KUKA KRL program: MyProgram_309().src

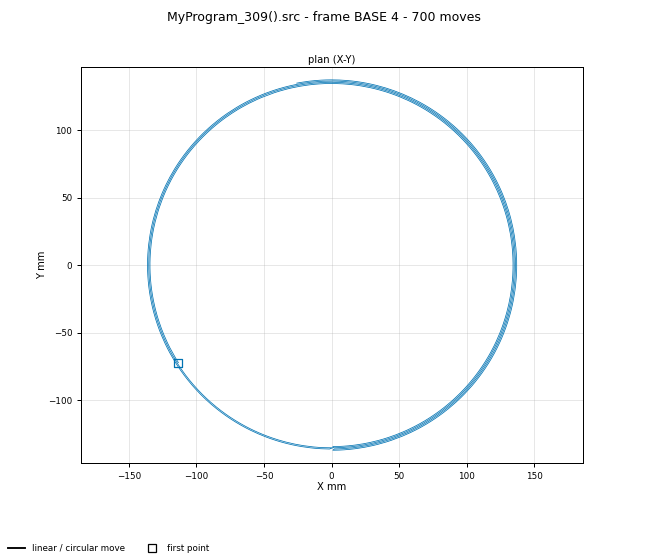
[picture p0: tool path of MyProgram_309().src in frame BASE 4, 700 of 700 moves have a stored position in this frame; points joined in program order, loops and branches not executed]
&ACCESS RVP
&REL 1
&PARAM TEMPLATE = C:\KRC\Roboter\Template\vorgabe
&PARAM EDITMASK = *
DEF MyProgram_309()
; ---- Setting reference (Base) ----
$BASE = BASE_DATA[4]

; --------------------------
; ---- Setting tool (TCP) ----
$TOOL = TOOL_DATA[3]
; --------------------------

$VEL.CP = VEL_APROX_PRINT
Startdeposition()
$VEL.CP = VEL_PRINT
LIN {X -113.3933,Y -72.2581,Z 182,A -144.0456,B 4.4589,C 0.2959,E1 4.3339,E2 236.7047} C_DIS
LIN {X -115.3766,Y -69.0471,Z 182,A -147.133,B 4.4585,C 0.3023,E1 4.3294,E2 239.9737} C_DIS
LIN {X -119.7006,Y -61.2412,Z 182,A -149.3934,B 4.4598,C 0.2824,E1 4.3266,E2 242.0427} C_DIS
LIN {X -121.551,Y -57.4829,Z 182,A -151.4804,B 4.46,C 0.28,E1 4.324,E2 244.1665} C_DIS
LIN {X -122.8459,Y -54.659,Z 182,A -152.8316,B 4.4602,C 0.2768,E1 4.3224,E2 245.5205} C_DIS
LIN {X -124.1948,Y -51.5211,Z 182,A -154.355,B 4.4604,C 0.2735,E1 4.3208,E2 247.0515} C_DIS
LIN {X -125.9546,Y -47.0544,Z 182,A -156.4644,B 4.4607,C 0.2686,E1 4.3186,E2 249.1678} C_DIS
LIN {X -127.2931,Y -43.3101,Z 182,A -158.1642,B 4.4609,C 0.2641,E1 4.3171,E2 250.8675} C_DIS
LIN {X -128.1422,Y -40.7223,Z 182,A -159.3873,B 4.4611,C 0.2614,E1 4.316,E2 252.0976} C_DIS
LIN {X -129.0534,Y -37.7348,Z 182,A -160.7492,B 4.4613,C 0.258,E1 4.3149,E2 253.4625} C_DIS
LIN {X -130.247,Y -33.3845,Z 182,A -162.5253,B 4.4616,C 0.2518,E1 4.3137,E2 255.2196} C_DIS
LIN {X -131.0025,Y -30.2853,Z 182,A -164.2358,B 4.4617,C 0.2504,E1 4.3125,E2 256.9725} C_DIS
LIN {X -131.9051,Y -26.083,Z 182,A -166.023,B 4.462,C 0.2451,E1 4.3115,E2 258.7533} C_DIS
LIN {X -132.6145,Y -22.1846,Z 182,A -167.7411,B 4.4623,C 0.2406,E1 4.3107,E2 260.4739} C_DIS
LIN {X -133.1933,Y -18.4034,Z 182,A -169.5897,B 4.4624,C 0.2374,E1 4.3099,E2 262.3483} C_DIS
LIN {X -133.6998,Y -14.2533,Z 182,A -171.2997,B 4.4627,C 0.2319,E1 4.3094,E2 264.0484} C_DIS
LIN {X -134.0654,Y -10.2705,Z 182,A -173.1645,B 4.4629,C 0.2282,E1 4.3089,E2 265.9317} C_DIS
LIN {X -134.3281,Y -5.9384,Z 182,A -174.9356,B 4.4632,C 0.2224,E1 4.3087,E2 267.6919} C_DIS
LIN {X -134.4379,Y -2.2975,Z 182,A -176.6146,B 4.4634,C 0.2188,E1 4.3085,E2 269.3853} C_DIS
LIN {X -134.4464,Y 1.7844,Z 182,A -178.4359,B 4.4636,C 0.2144,E1 4.3085,E2 271.2154} C_DIS
LIN {X -134.354,Y 5.2733,Z 182,A -179.936,B 4.4638,C 0.2103,E1 4.3087,E2 272.716} C_DIS
LIN {X -134.1215,Y 9.5026,Z 182,A 178.1862,B 4.464,C 0.2057,E1 4.309,E2 274.6013} C_DIS
LIN {X -133.8199,Y 13.0792,Z 182,A 176.6504,B 4.4642,C 0.2014,E1 4.3094,E2 276.1368} C_DIS
LIN {X -133.502,Y 15.9997,Z 182,A 175.3587,B 4.4643,C 0.1981,E1 4.3098,E2 277.4323} C_DIS
LIN {X -133.023,Y 19.5953,Z 182,A 173.6191,B 4.4645,C 0.195,E1 4.3105,E2 279.1944} C_DIS
LIN {X -132.3689,Y 23.6053,Z 182,A 171.9298,B 4.4647,C 0.1899,E1 4.3113,E2 280.8772} C_DIS
LIN {X -131.671,Y 27.2336,Z 182,A 170.256,B 4.4649,C 0.1861,E1 4.3122,E2 282.5618} C_DIS
LIN {X -130.5324,Y 32.2586,Z 182,A 168.0955,B 4.4651,C 0.1799,E1 4.3136,E2 284.7163} C_DIS
LIN {X -129.2234,Y 37.1542,Z 182,A 165.915,B 4.4653,C 0.1741,E1 4.3152,E2 286.8977} C_DIS
LIN {X -128.5071,Y 39.5558,Z 182,A 164.7164,B 4.4654,C 0.172,E1 4.3162,E2 288.1112} C_DIS
LIN {X -127.5833,Y 42.4406,Z 182,A 163.3928,B 4.4655,C 0.1687,E1 4.3173,E2 289.4377} C_DIS
LIN {X -126.1534,Y 46.5237,Z 182,A 161.5675,B 4.4657,C 0.1637,E1 4.319,E2 291.2594} C_DIS
LIN {X -125.1691,Y 49.1075,Z 182,A 160.3104,B 4.4658,C 0.1611,E1 4.3203,E2 292.525} C_DIS
LIN {X -123.9551,Y 52.095,Z 182,A 158.8275,B 4.4659,C 0.1582,E1 4.3219,E2 294.0197} C_DIS
LIN {X -122.5618,Y 55.2941,Z 182,A 157.3536,B 4.4661,C 0.1543,E1 4.3236,E2 295.4909} C_DIS
LIN {X -121.0569,Y 58.5172,Z 182,A 155.4896,B 4.4661,C 0.1527,E1 4.3259,E2 297.3955} C_DIS
LIN {X -118.7591,Y 63.0499,Z 182,A 153.5389,B 4.4664,C 0.1458,E1 4.3283,E2 299.3186} C_DIS
LIN {X -116.7267,Y 66.7391,Z 182,A 151.5986,B 4.4664,C 0.1424,E1 4.331,E2 301.275} C_DIS
LIN {X -114.4006,Y 70.6531,Z 182,A 149.1045,B 4.4664,C 0.1414,E1 4.3347,E2 303.8333} C_DIS
LIN {X -111.8542,Y 74.6179,Z 182,A 147.5238,B 4.4667,C 0.1338,E1 4.3371,E2 305.3616} C_DIS
LIN {X -109.1703,Y 78.493,Z 182,A 145.5025,B 4.4669,C 0.1293,E1 4.3403,E2 307.3828} C_DIS
LIN {X -106.7613,Y 81.7387,Z 182,A 143.725,B 4.4669,C 0.1258,E1 4.3433,E2 309.1654} C_DIS
LIN {X -104.0626,Y 85.1479,Z 182,A 141.8241,B 4.4671,C 0.122,E1 4.3467,E2 311.0705} C_DIS
LIN {X -101.1349,Y 88.6059,Z 182,A 139.8527,B 4.4671,C 0.1182,E1 4.3503,E2 313.0452} C_DIS
LIN {X -98.1961,Y 91.8521,Z 182,A 137.9249,B 4.4673,C 0.1148,E1 4.3539,E2 314.9788} C_DIS
LIN {X -95.323,Y 94.83,Z 182,A 136.1391,B 4.4673,C 0.1114,E1 4.3574,E2 316.7659} C_DIS
LIN {X -92.1703,Y 97.8971,Z 182,A 134.199,B 4.4674,C 0.1083,E1 4.3613,E2 318.7124} C_DIS
LIN {X -88.8308,Y 100.9375,Z 182,A 132.2757,B 4.4675,C 0.1047,E1 4.3653,E2 320.634} C_DIS
LIN {X -85.661,Y 103.6407,Z 182,A 130.4375,B 4.4675,C 0.102,E1 4.3693,E2 322.4783} C_DIS
LIN {X -82.322,Y 106.3122,Z 182,A 128.5912,B 4.4676,C 0.099,E1 4.3733,E2 324.3259} C_DIS
LIN {X -78.8871,Y 108.8854,Z 182,A 126.7591,B 4.4676,C 0.096,E1 4.3775,E2 326.1571} C_DIS
LIN {X -73.7106,Y 112.4545,Z 182,A 123.4758,B 4.4676,C 0.0965,E1 4.3852,E2 329.5096} C_DIS
LIN {X -69.7248,Y 114.9682,Z 182,A 122.124,B 4.4679,C 0.0886,E1 4.3883,E2 330.7825} C_DIS
LIN {X -66.9003,Y 116.6347,Z 182,A 120.1078,B 4.4678,C 0.0914,E1 4.3933,E2 332.8708} C_DIS
LIN {X -63.1989,Y 118.6809,Z 182,A 118.798,B 4.4679,C 0.0852,E1 4.3964,E2 334.1213} C_DIS
LIN {X -61.0835,Y 119.7809,Z 182,A 117.6379,B 4.4679,C 0.0852,E1 4.3993,E2 335.2977} C_DIS
LIN {X -57.3839,Y 121.5983,Z 182,A 115.9821,B 4.4679,C 0.0822,E1 4.4034,E2 336.9403} C_DIS
LIN {X -54.881,Y 122.7466,Z 182,A 114.6943,B 4.4679,C 0.0818,E1 4.4068,E2 338.2408} C_DIS
LIN {X -51.5957,Y 124.1636,Z 182,A 113.1875,B 4.468,C 0.0801,E1 4.4106,E2 339.7446} C_DIS
LIN {X -42.4267,Y 127.5879,Z 182,A 108.5492,B 4.468,C 0.0801,E1 4.423,E2 344.4352} C_DIS
LIN {X -38.4167,Y 128.8538,Z 182,A 107.2755,B 4.4681,C 0.0745,E1 4.4262,E2 345.6469} C_DIS
LIN {X -35.4991,Y 129.6884,Z 182,A 105.9279,B 4.4681,C 0.074,E1 4.4298,E2 347.0002} C_DIS
LIN {X -32.7166,Y 130.4165,Z 182,A 104.7062,B 4.4681,C 0.0732,E1 4.4331,E2 348.2206} C_DIS
LIN {X -29.8649,Y 131.0985,Z 182,A 103.3874,B 4.4681,C 0.0731,E1 4.4367,E2 349.5468} C_DIS
LIN {X -26.0554,Y 131.9107,Z 182,A 101.7586,B 4.4681,C 0.0719,E1 4.4412,E2 351.1712} C_DIS
LIN {X -23.3572,Y 132.4133,Z 182,A 100.6147,B 4.4681,C 0.0712,E1 4.4443,E2 352.3113} C_DIS
LIN {X -19.9287,Y 132.9738,Z 182,A 99.0996,B 4.4681,C 0.071,E1 4.4485,E2 353.8298} C_DIS
LIN {X -16.7934,Y 133.4062,Z 182,A 97.2359,B 4.4681,C 0.0751,E1 4.4538,E2 355.7534} C_DIS
LIN {X -12.6819,Y 133.858,Z 182,A 95.9309,B 4.4681,C 0.0707,E1 4.4573,E2 357.0037} C_DIS
LIN {X -9.5581,Y 134.1174,Z 182,A 94.5437,B 4.4681,C 0.0709,E1 4.4612,E2 358.3963} C_DIS
LIN {X -5.5166,Y 134.3445,Z 182,A 92.8589,B 4.4681,C 0.0704,E1 4.4659,E2 360.0755} C_DIS
LIN {X -1.4978,Y 134.4505,Z 182,A 91.015,B 4.4681,C 0.0717,E1 4.4711,E2 361.9342} C_DIS
LIN {X 2.3924,Y 134.4363,Z 182,A 89.4627,B 4.4681,C 0.0708,E1 4.4754,E2 363.4733} C_DIS
LIN {X 5.8114,Y 134.333,Z 182,A 88.1347,B 4.4681,C 0.0699,E1 4.479,E2 364.7854} C_DIS
LIN {X 8.5441,Y 134.1859,Z 182,A 86.7961,B 4.4681,C 0.0718,E1 4.4828,E2 366.1439} C_DIS
LIN {X 13.4353,Y 133.7857,Z 182,A 84.7941,B 4.4681,C 0.0716,E1 4.4884,E2 368.1346} C_DIS
LIN {X 17.4287,Y 133.3229,Z 182,A 83.0133,B 4.4681,C 0.0729,E1 4.4933,E2 369.9227} C_DIS
LIN {X 22.1823,Y 132.6148,Z 182,A 81.0965,B 4.4681,C 0.0727,E1 4.4986,E2 371.8234} C_DIS
LIN {X 25.2731,Y 132.0606,Z 182,A 79.7667,B 4.4681,C 0.0734,E1 4.5022,E2 373.1518} C_DIS
LIN {X 28.5205,Y 131.3976,Z 182,A 78.3441,B 4.4681,C 0.0744,E1 4.5061,E2 374.5753} C_DIS
LIN {X 32.4205,Y 130.4917,Z 182,A 76.5461,B 4.4681,C 0.0765,E1 4.511,E2 376.3837} C_DIS
LIN {X 36.0959,Y 129.5215,Z 182,A 74.531,B 4.468,C 0.0819,E1 4.5166,E2 378.445} C_DIS
LIN {X 40.4003,Y 128.2448,Z 182,A 73.2819,B 4.468,C 0.0768,E1 4.5197,E2 379.6153} C_DIS
LIN {X 43.736,Y 127.1454,Z 182,A 71.5814,B 4.468,C 0.0803,E1 4.5243,E2 381.3396} C_DIS
LIN {X 47.3865,Y 125.8303,Z 182,A 70.0326,B 4.468,C 0.0809,E1 4.5283,E2 382.8757} C_DIS
LIN {X 50.52,Y 124.6053,Z 182,A 68.6167,B 4.468,C 0.0823,E1 4.532,E2 384.2893} C_DIS
LIN {X 54.1914,Y 123.0551,Z 182,A 66.9764,B 4.468,C 0.0837,E1 4.5362,E2 385.9226} C_DIS
LIN {X 56.6157,Y 121.9564,Z 182,A 65.8155,B 4.468,C 0.0854,E1 4.5391,E2 387.0865} C_DIS
LIN {X 59.7801,Y 120.4371,Z 182,A 64.3292,B 4.4679,C 0.0872,E1 4.5428,E2 388.5715} C_DIS
LIN {X 63.1887,Y 118.6862,Z 182,A 62.8242,B 4.4679,C 0.0881,E1 4.5465,E2 390.0613} C_DIS
LIN {X 66.3073,Y 116.9729,Z 182,A 61.1293,B 4.4678,C 0.0922,E1 4.5507,E2 391.7774} C_DIS
LIN {X 69.8955,Y 114.8649,Z 182,A 59.4108,B 4.4678,C 0.0943,E1 4.5548,E2 393.4893} C_DIS
LIN {X 73.1101,Y 112.8456,Z 182,A 57.8239,B 4.4677,C 0.0964,E1 4.5586,E2 395.0726} C_DIS
LIN {X 76.8735,Y 110.3162,Z 182,A 55.9392,B 4.4677,C 0.0991,E1 4.5629,E2 396.9517} C_DIS
LIN {X 80.1605,Y 107.9515,Z 182,A 54.2252,B 4.4676,C 0.1019,E1 4.5667,E2 398.6644} C_DIS
LIN {X 83.4929,Y 105.3956,Z 182,A 52.5057,B 4.4676,C 0.1043,E1 4.5705,E2 400.3757} C_DIS
LIN {X 86.7231,Y 102.7543,Z 182,A 50.7346,B 4.4674,C 0.1075,E1 4.5743,E2 402.1461} C_DIS
LIN {X 90.7436,Y 99.2215,Z 182,A 48.5047,B 4.4674,C 0.1113,E1 4.579,E2 404.3703} C_DIS
LIN {X 93.9259,Y 96.2144,Z 182,A 46.66,B 4.4673,C 0.1148,E1 4.5827,E2 406.2127} C_DIS
LIN {X 97.2485,Y 92.8543,Z 182,A 44.8621,B 4.4673,C 0.1164,E1 4.5861,E2 407.9851} C_DIS
LIN {X 99.7983,Y 90.1088,Z 182,A 43.1522,B 4.4671,C 0.1211,E1 4.5894,E2 409.709} C_DIS
LIN {X 102.7253,Y 86.7572,Z 182,A 41.3372,B 4.4671,C 0.1243,E1 4.5927,E2 411.5147} C_DIS
LIN {X 105.486,Y 83.379,Z 182,A 39.4855,B 4.4669,C 0.1283,E1 4.5959,E2 413.366} C_DIS
LIN {X 107.6526,Y 80.5619,Z 182,A 38.1164,B 4.4669,C 0.13,E1 4.5982,E2 414.718} C_DIS
LIN {X 110.0357,Y 77.2749,Z 182,A 36.3306,B 4.4667,C 0.1347,E1 4.6011,E2 416.5112} C_DIS
LIN {X 112.198,Y 74.1002,Z 182,A 34.758,B 4.4667,C 0.1378,E1 4.6035,E2 418.0765} C_DIS
LIN {X 114.3595,Y 70.7194,Z 182,A 33.0845,B 4.4665,C 0.1415,E1 4.606,E2 419.7462} C_DIS
LIN {X 116.2486,Y 67.5685,Z 182,A 31.557,B 4.4664,C 0.1449,E1 4.6082,E2 421.2697} C_DIS
LIN {X 118.4291,Y 63.6691,Z 182,A 29.7729,B 4.4663,C 0.1482,E1 4.6106,E2 423.0401} C_DIS
LIN {X 119.8546,Y 60.9386,Z 182,A 28.4894,B 4.4662,C 0.1511,E1 4.6122,E2 424.3205} C_DIS
LIN {X 121.6394,Y 57.298,Z 182,A 26.8491,B 4.4661,C 0.1545,E1 4.6142,E2 425.951} C_DIS
LIN {X 122.7451,Y 54.8845,Z 182,A 25.7578,B 4.466,C 0.1569,E1 4.6154,E2 427.0379} C_DIS
LIN {X 124.9219,Y 49.7342,Z 182,A 23.1326,B 4.4656,C 0.1662,E1 4.6182,E2 429.6938} C_DIS
LIN {X 126.1191,Y 46.6154,Z 182,A 22.0493,B 4.4656,C 0.1657,E1 4.6193,E2 430.7365} C_DIS
LIN {X 127.1406,Y 43.7499,Z 182,A 20.7434,B 4.4656,C 0.1693,E1 4.6205,E2 432.0441} C_DIS
LIN {X 128.3104,Y 40.1957,Z 182,A 19.2597,B 4.4654,C 0.1722,E1 4.6217,E2 433.5152} C_DIS
LIN {X 129.3835,Y 36.5893,Z 182,A 17.6578,B 4.4652,C 0.1766,E1 4.623,E2 435.1177} C_DIS
LIN {X 130.3423,Y 33.0092,Z 182,A 16.1637,B 4.4652,C 0.1798,E1 4.624,E2 436.6024} C_DIS
LIN {X 131.1561,Y 29.6128,Z 182,A 14.671,B 4.4649,C 0.184,E1 4.625,E2 438.0965} C_DIS
LIN {X 131.8816,Y 26.1986,Z 182,A 13.2924,B 4.4649,C 0.1868,E1 4.6257,E2 439.4627} C_DIS
LIN {X 132.435,Y 23.2362,Z 182,A 12.0709,B 4.4647,C 0.1896,E1 4.6263,E2 440.6772} C_DIS
LIN {X 132.9509,Y 20.0765,Z 182,A 10.6053,B 4.4645,C 0.1947,E1 4.627,E2 442.1561} C_DIS
LIN {X 133.4213,Y 16.6763,Z 182,A 9.3253,B 4.4645,C 0.1965,E1 4.6274,E2 443.4147} C_DIS
LIN {X 133.7277,Y 13.9936,Z 182,A 8.2364,B 4.4643,C 0.1989,E1 4.6278,E2 444.4967} C_DIS
LIN {X 134.0514,Y 10.4624,Z 182,A 6.6919,B 4.4641,C 0.2036,E1 4.6281,E2 446.0464} C_DIS
LIN {X 134.3161,Y 6.1891,Z 182,A 4.7647,B 4.4638,C 0.2101,E1 4.6284,E2 447.9875} C_DIS
LIN {X 134.4515,Y 1.4573,Z 182,A 2.9283,B 4.4636,C 0.2135,E1 4.6285,E2 449.8031} C_DIS
LIN {X 134.4277,Y -2.9093,Z 182,A 1.2197,B 4.4635,C 0.2169,E1 4.6285,E2 451.4941} C_DIS
LIN {X 134.2584,Y -7.3369,Z 182,A -0.614,B 4.4632,C 0.2215,E1 4.6283,E2 453.3225} C_DIS
LIN {X 133.9862,Y -11.2465,Z 182,A -2.334,B 4.463,C 0.2269,E1 4.6279,E2 455.0498} C_DIS
LIN {X 133.6364,Y -14.8426,Z 182,A -3.7012,B 4.4629,C 0.229,E1 4.6275,E2 456.3969} C_DIS
LIN {X 133.2626,Y -17.8893,Z 182,A -5.1369,B 4.4626,C 0.2344,E1 4.627,E2 457.8494} C_DIS
LIN {X 132.5488,Y -22.5782,Z 182,A -6.9217,B 4.4624,C 0.237,E1 4.6262,E2 459.6064} C_DIS
LIN {X 131.9195,Y -26.0115,Z 182,A -8.3947,B 4.4622,C 0.241,E1 4.6254,E2 461.0789} C_DIS
LIN {X 131.2851,Y -29.0417,Z 182,A -9.6737,B 4.4621,C 0.2442,E1 4.6247,E2 462.3539} C_DIS
LIN {X 130.6233,Y -31.8813,Z 182,A -10.8534,B 4.4619,C 0.2468,E1 4.6239,E2 463.5267} C_DIS
LIN {X 129.8554,Y -34.8762,Z 182,A -12.2063,B 4.4617,C 0.2509,E1 4.623,E2 464.8851} C_DIS
LIN {X 128.6748,Y -39.008,Z 182,A -13.9853,B 4.4614,C 0.2553,E1 4.6216,E2 466.6591} C_DIS
LIN {X 127.1875,Y -43.6146,Z 182,A -15.9399,B 4.4612,C 0.2595,E1 4.6199,E2 468.6019} C_DIS
LIN {X 126.027,Y -46.8614,Z 182,A -17.5288,B 4.4609,C 0.2649,E1 4.6183,E2 470.2069} C_DIS
LIN {X 124.5326,Y -50.7002,Z 182,A -19.1914,B 4.4607,C 0.2684,E1 4.6166,E2 471.8594} C_DIS
LIN {X 123.1292,Y -54.0221,Z 182,A -20.5599,B 4.4606,C 0.2704,E1 4.6151,E2 473.2082} C_DIS
LIN {X 121.8799,Y -56.7812,Z 182,A -21.9042,B 4.4603,C 0.2744,E1 4.6136,E2 474.5602} C_DIS
LIN {X 120.3627,Y -59.9308,Z 182,A -23.2834,B 4.4602,C 0.2769,E1 4.6119,E2 475.9268} C_DIS
LIN {X 118.0655,Y -64.3408,Z 182,A -25.3175,B 4.4599,C 0.2812,E1 4.6092,E2 477.9522} C_DIS
LIN {X 116.1605,Y -67.7206,Z 182,A -27.0291,B 4.4596,C 0.2861,E1 4.6069,E2 479.6725} C_DIS
LIN {X 114.0228,Y -71.2606,Z 182,A -28.7623,B 4.4593,C 0.29,E1 4.6043,E2 481.4035} C_DIS
LIN {X 111.6949,Y -74.8566,Z 182,A -30.5206,B 4.4591,C 0.2936,E1 4.6016,E2 483.155} C_DIS
LIN {X 109.3703,Y -78.2134,Z 182,A -32.2078,B 4.4589,C 0.2971,E1 4.5989,E2 484.837} C_DIS
LIN {X 106.689,Y -81.8333,Z 182,A -34.0857,B 4.4586,C 0.301,E1 4.5958,E2 486.7113} C_DIS
LIN {X 104.0053,Y -85.2181,Z 182,A -35.8735,B 4.4584,C 0.3046,E1 4.5927,E2 488.494} C_DIS
LIN {X 100.7335,Y -89.0616,Z 182,A -37.7925,B 4.4582,C 0.3065,E1 4.5892,E2 490.3856} C_DIS
LIN {X 98.2774,Y -91.7648,Z 182,A -39.4623,B 4.4579,C 0.3112,E1 4.586,E2 492.071} C_DIS
LIN {X 95.1977,Y -94.9561,Z 182,A -41.3675,B 4.4576,C 0.3154,E1 4.5823,E2 493.9798} C_DIS
LIN {X 91.2794,Y -98.729,Z 182,A -43.4698,B 4.4575,C 0.3175,E1 4.5781,E2 496.0567} C_DIS
LIN {X 88.6795,Y -101.0706,Z 182,A -45.1059,B 4.4571,C 0.3222,E1 4.5746,E2 497.7125} C_DIS
LIN {X 85.3767,Y -103.8756,Z 182,A -46.8502,B 4.457,C 0.3245,E1 4.5709,E2 499.4453} C_DIS
LIN {X 82.3404,Y -106.298,Z 182,A -48.4788,B 4.4568,C 0.3272,E1 4.5673,E2 501.0719} C_DIS
LIN {X 79.5563,Y -108.3974,Z 182,A -49.8643,B 4.4566,C 0.3287,E1 4.5643,E2 502.4459} C_DIS
LIN {X 76.4279,Y -110.6261,Z 182,A -51.562,B 4.4564,C 0.3322,E1 4.5604,E2 504.1526} C_DIS
LIN {X 72.8163,Y -113.0359,Z 182,A -53.3398,B 4.4562,C 0.3344,E1 4.5562,E2 505.9227} C_DIS
LIN {X 69.2003,Y -115.2851,Z 182,A -55.1591,B 4.456,C 0.3373,E1 4.5519,E2 507.744} C_DIS
LIN {X 65.4541,Y -117.4525,Z 182,A -56.9794,B 4.4558,C 0.3398,E1 4.5475,E2 509.5626} C_DIS
LIN {X 61.3924,Y -119.6236,Z 182,A -58.6597,B 4.4558,C 0.3394,E1 4.5434,E2 511.2085} C_DIS
LIN {X 58.673,Y -120.9825,Z 182,A -60.0649,B 4.4556,C 0.3424,E1 4.5398,E2 512.6287} C_DIS
LIN {X 56.3839,Y -122.0636,Z 182,A -61.2344,B 4.4554,C 0.3449,E1 4.5369,E2 513.8104} C_DIS
LIN {X 52.8908,Y -123.6183,Z 182,A -63.5089,B 4.4547,C 0.3541,E1 4.5308,E2 516.1677} C_DIS
LIN {X 47.5793,Y -125.7581,Z 182,A -65.014,B 4.4553,C 0.3465,E1 4.5272,E2 517.5561} C_DIS
LIN {X 42.1713,Y -127.6729,Z 182,A -67.5798,B 4.455,C 0.3505,E1 4.5204,E2 520.1391} C_DIS
LIN {X 38.1773,Y -128.9239,Z 182,A -69.4257,B 4.4548,C 0.3528,E1 4.5154,E2 521.9942} C_DIS
LIN {X 34.3309,Y -130.0008,Z 182,A -71.0744,B 4.4548,C 0.3537,E1 4.511,E2 523.6372} C_DIS
LIN {X 30.9344,Y -130.8515,Z 182,A -72.4808,B 4.4548,C 0.354,E1 4.5072,E2 525.0336} C_DIS
LIN {X 28.1939,Y -131.4681,Z 182,A -73.6699,B 4.4546,C 0.3548,E1 4.5039,E2 526.2224} C_DIS
LIN {X 23.3364,Y -132.4171,Z 182,A -75.7501,B 4.4546,C 0.3559,E1 4.4983,E2 528.3002} C_DIS
LIN {X 19.8941,Y -132.9791,Z 182,A -77.228,B 4.4546,C 0.3567,E1 4.4942,E2 529.778} C_DIS
LIN {X 17.3536,Y -133.3328,Z 182,A -78.4563,B 4.4543,C 0.3586,E1 4.4907,E2 531.024} C_DIS
LIN {X 12.3919,Y -133.8859,Z 182,A -80.9068,B 4.454,C 0.3628,E1 4.4838,E2 533.5168} C_DIS
LIN {X 8.4264,Y -134.1932,Z 182,A -82.1981,B 4.4543,C 0.3593,E1 4.4803,E2 534.7576} C_DIS
LIN {X 4.743,Y -134.3747,Z 182,A -83.6718,B 4.4543,C 0.3587,E1 4.4762,E2 536.2197} C_DIS
LIN {X 0.9641,Y -134.4524,Z 182,A -85.5454,B 4.4541,C 0.3616,E1 4.4709,E2 538.1275} C_DIS
Enddeposition()
LIN {X 0.9641,Y -134.4524,Z 182,A -85.5454,B 4.4541,C 0.3616,E1 4.4709,E2 538.1275} C_DIS
Startdeposition()
$VEL.CP = VEL_PRINT
LIN {X 1.5996,Y -135.3511,Z 182,A -84.3043,B 4.4548,C 0.3542,E1 4.4748,E2 536.7934} C_DIS
LIN {X 8.4271,Y -135.0963,Z 182,A -81.4838,B 4.4548,C 0.3542,E1 4.4826,E2 533.9808} C_DIS
LIN {X 15.2303,Y -134.5013,Z 182,A -78.6391,B 4.4548,C 0.3535,E1 4.4905,E2 531.1406} C_DIS
LIN {X 18.8912,Y -134.0342,Z 182,A -77.0659,B 4.4548,C 0.3526,E1 4.4948,E2 529.5651} C_DIS
LIN {X 23.0843,Y -133.378,Z 182,A -75.0501,B 4.4552,C 0.3492,E1 4.5005,E2 527.5198} C_DIS
LIN {X 28.2212,Y -132.3845,Z 182,A -73.118,B 4.455,C 0.3507,E1 4.5057,E2 525.623} C_DIS
LIN {X 31.6043,Y -131.6174,Z 182,A -71.686,B 4.455,C 0.35,E1 4.5095,E2 524.1948} C_DIS
LIN {X 34.9586,Y -130.7664,Z 182,A -70.192,B 4.4552,C 0.3484,E1 4.5136,E2 522.6961} C_DIS
LIN {X 38.6291,Y -129.7309,Z 182,A -68.4986,B 4.4554,C 0.3461,E1 4.5182,E2 520.9914} C_DIS
LIN {X 42.4486,Y -128.5307,Z 182,A -66.9042,B 4.4554,C 0.3455,E1 4.5224,E2 519.4089} C_DIS
LIN {X 46.6809,Y -127.057,Z 182,A -64.7935,B 4.4558,C 0.341,E1 4.528,E2 517.2691} C_DIS
LIN {X 53.5716,Y -124.3061,Z 182,A -61.9854,B 4.4558,C 0.341,E1 4.5352,E2 514.5021} C_DIS
LIN {X 56.4713,Y -123.0164,Z 182,A -60.6059,B 4.4559,C 0.339,E1 4.5387,E2 513.1169} C_DIS
LIN {X 59.9731,Y -121.3471,Z 182,A -58.9333,B 4.4561,C 0.3364,E1 4.5429,E2 511.4391} C_DIS
LIN {X 64.1801,Y -119.1779,Z 182,A -56.9422,B 4.4563,C 0.3337,E1 4.5478,E2 509.4482} C_DIS
LIN {X 68.029,Y -117.0237,Z 182,A -55.0992,B 4.4565,C 0.3311,E1 4.5523,E2 507.6069} C_DIS
LIN {X 71.5627,Y -114.8965,Z 182,A -53.391,B 4.4567,C 0.3288,E1 4.5563,E2 505.9022} C_DIS
LIN {X 75.3973,Y -112.4178,Z 182,A -51.4833,B 4.4569,C 0.3259,E1 4.5608,E2 503.9962} C_DIS
LIN {X 79.1242,Y -109.8268,Z 182,A -49.7404,B 4.457,C 0.3247,E1 4.5647,E2 502.2749} C_DIS
LIN {X 82.5708,Y -107.2598,Z 182,A -47.7844,B 4.4574,C 0.3198,E1 4.5691,E2 500.2997} C_DIS
LIN {X 86.2159,Y -104.3516,Z 182,A -45.9123,B 4.4575,C 0.3173,E1 4.5731,E2 498.4391} C_DIS
LIN {X 89.5705,Y -101.4868,Z 182,A -44.27,B 4.4575,C 0.3164,E1 4.5766,E2 496.8244} C_DIS
LIN {X 94.6889,Y -96.7288,Z 182,A -41.2137,B 4.4581,C 0.3093,E1 4.5828,E2 493.7531} C_DIS
LIN {X 97.692,Y -93.695,Z 182,A -39.4079,B 4.4584,C 0.3055,E1 4.5863,E2 491.9459} C_DIS
LIN {X 99.7683,Y -91.4808,Z 182,A -37.6652,B 4.4589,C 0.297,E1 4.5897,E2 490.1428} C_DIS
LIN {X 103.0191,Y -87.8039,Z 182,A -36.1339,B 4.4588,C 0.2992,E1 4.5924,E2 488.6805} C_DIS
LIN {X 105.7456,Y -84.5007,Z 182,A -34.3899,B 4.459,C 0.296,E1 4.5954,E2 486.9439} C_DIS
LIN {X 108.1621,Y -81.3844,Z 182,A -32.7772,B 4.4592,C 0.2928,E1 4.5982,E2 485.3371} C_DIS
LIN {X 110.7077,Y -77.8862,Z 182,A -30.9529,B 4.4595,C 0.2886,E1 4.6011,E2 483.5121} C_DIS
LIN {X 113.2845,Y -74.0893,Z 182,A -29.0317,B 4.4598,C 0.2842,E1 4.6041,E2 481.5919} C_DIS
LIN {X 115.6228,Y -70.3844,Z 182,A -27.2329,B 4.46,C 0.2803,E1 4.6067,E2 479.7987} C_DIS
LIN {X 117.8953,Y -66.5069,Z 182,A -25.4078,B 4.4602,C 0.2766,E1 4.6093,E2 477.9819} C_DIS
LIN {X 121.4888,Y -59.6858,Z 182,A -22.379,B 4.4606,C 0.2712,E1 4.6131,E2 474.9804} C_DIS
LIN {X 122.8351,Y -56.8632,Z 182,A -21.0692,B 4.4608,C 0.268,E1 4.6147,E2 473.6713} C_DIS
LIN {X 124.0339,Y -54.2012,Z 182,A -19.8,B 4.461,C 0.2643,E1 4.6161,E2 472.3968} C_DIS
LIN {X 125.4634,Y -50.8023,Z 182,A -17.9063,B 4.4615,C 0.2559,E1 4.6182,E2 470.4591} C_DIS
LIN {X 126.9388,Y -46.9969,Z 182,A -16.0641,B 4.4618,C 0.2497,E1 4.62,E2 468.6007} C_DIS
LIN {X 128.5648,Y -42.3462,Z 182,A -14.5273,B 4.4618,C 0.2512,E1 4.6213,E2 467.1326} C_DIS
LIN {X 129.8144,Y -38.3441,Z 182,A -12.8677,B 4.4619,C 0.2478,E1 4.6226,E2 465.4862} C_DIS
LIN {X 130.744,Y -35.0425,Z 182,A -11.5095,B 4.4621,C 0.245,E1 4.6236,E2 464.1388} C_DIS
LIN {X 131.6157,Y -31.6111,Z 182,A -10.0169,B 4.4623,C 0.241,E1 4.6246,E2 462.6457} C_DIS
LIN {X 132.4712,Y -27.8193,Z 182,A -8.3148,B 4.4626,C 0.2357,E1 4.6256,E2 460.9352} C_DIS
LIN {X 133.2488,Y -23.8063,Z 182,A -6.2362,B 4.4631,C 0.2263,E1 4.6267,E2 458.8107} C_DIS
LIN {X 133.991,Y -19.194,Z 182,A -4.8326,B 4.463,C 0.2282,E1 4.6272,E2 457.4787} C_DIS
LIN {X 134.4975,Y -15.2649,Z 182,A -3.2105,B 4.4632,C 0.2242,E1 4.6277,E2 455.8624} C_DIS
LIN {X 134.849,Y -11.7426,Z 182,A -1.9631,B 4.4632,C 0.2232,E1 4.6281,E2 454.6455} C_DIS
LIN {X 135.1158,Y -8.1112,Z 182,A 0.1342,B 4.4638,C 0.2116,E1 4.6284,E2 452.4766} C_DIS
LIN {X 135.2981,Y -4.0681,Z 182,A 1.3946,B 4.4638,C 0.2126,E1 4.6286,E2 451.2724} C_DIS
LIN {X 135.3603,Y -0.3013,Z 182,A 2.8763,B 4.4638,C 0.2095,E1 4.6286,E2 449.8039} C_DIS
LIN {X 135.2462,Y 5.5297,Z 182,A 5.6192,B 4.4644,C 0.199,E1 4.6284,E2 447.0245} C_DIS
LIN {X 135.0582,Y 9.041,Z 182,A 6.7677,B 4.4644,C 0.1992,E1 4.6282,E2 445.918} C_DIS
LIN {X 134.7909,Y 12.3981,Z 182,A 8.1579,B 4.4645,C 0.1956,E1 4.6278,E2 444.5313} C_DIS
LIN {X 134.4168,Y 15.9418,Z 182,A 9.9465,B 4.4649,C 0.1877,E1 4.6273,E2 442.7063} C_DIS
LIN {X 133.9308,Y 19.6153,Z 182,A 11.2046,B 4.4649,C 0.1873,E1 4.6268,E2 441.4864} C_DIS
LIN {X 133.279,Y 23.6374,Z 182,A 12.7048,B 4.4649,C 0.1854,E1 4.6261,E2 440.0132} C_DIS
LIN {X 132.6493,Y 26.947,Z 182,A 14.1235,B 4.4651,C 0.1815,E1 4.6253,E2 438.5946} C_DIS
LIN {X 132.0075,Y 29.9336,Z 182,A 15.45,B 4.4653,C 0.1775,E1 4.6245,E2 437.2631} C_DIS
LIN {X 131.2232,Y 33.2029,Z 182,A 16.7746,B 4.4653,C 0.1749,E1 4.6236,E2 435.95} C_DIS
LIN {X 130.3772,Y 36.3829,Z 182,A 18.1089,B 4.4655,C 0.1718,E1 4.6227,E2 434.6222} C_DIS
LIN {X 129.5927,Y 39.0892,Z 182,A 19.3423,B 4.4656,C 0.168,E1 4.6217,E2 433.3831} C_DIS
LIN {X 128.4695,Y 42.6323,Z 182,A 20.8365,B 4.4658,C 0.1648,E1 4.6204,E2 431.8979} C_DIS
LIN {X 127.2739,Y 46.0792,Z 182,A 22.3346,B 4.4658,C 0.1613,E1 4.619,E2 430.4047} C_DIS
LIN {X 126.139,Y 49.1006,Z 182,A 23.8843,B 4.4661,C 0.1553,E1 4.6174,E2 428.8315} C_DIS
LIN {X 123.9187,Y 54.4676,Z 182,A 26.1424,B 4.4662,C 0.1514,E1 4.615,E2 426.5972} C_DIS
LIN {X 122.2227,Y 58.1682,Z 182,A 27.6302,B 4.4662,C 0.1499,E1 4.6133,E2 425.1378} C_DIS
LIN {X 120.8252,Y 61.0192,Z 182,A 29.0988,B 4.4664,C 0.145,E1 4.6114,E2 423.6532} C_DIS
LIN {X 118.9462,Y 64.6088,Z 182,A 30.7903,B 4.4666,C 0.1409,E1 4.6092,E2 421.9639} C_DIS
LIN {X 116.7631,Y 68.475,Z 182,A 32.5909,B 4.4666,C 0.1373,E1 4.6067,E2 420.1724} C_DIS
LIN {X 114.5998,Y 72.0373,Z 182,A 34.3503,B 4.4668,C 0.1331,E1 4.6041,E2 418.413} C_DIS
LIN {X 112.3075,Y 75.5618,Z 182,A 36.0928,B 4.4669,C 0.1293,E1 4.6014,E2 416.6745} C_DIS
LIN {X 109.7648,Y 79.2098,Z 182,A 37.924,B 4.467,C 0.1255,E1 4.5985,E2 414.8489} C_DIS
LIN {X 107.477,Y 82.2868,Z 182,A 39.5695,B 4.4671,C 0.1216,E1 4.5957,E2 413.2002} C_DIS
LIN {X 104.4406,Y 86.1085,Z 182,A 41.5523,B 4.4672,C 0.118,E1 4.5922,E2 411.2271} C_DIS
LIN {X 101.3968,Y 89.6722,Z 182,A 43.4232,B 4.4673,C 0.1151,E1 4.5888,E2 409.3697} C_DIS
LIN {X 98.4313,Y 92.9177,Z 182,A 45.586,B 4.4675,C 0.1076,E1 4.5846,E2 407.1692} C_DIS
LIN {X 95.5992,Y 95.8295,Z 182,A 46.9468,B 4.4675,C 0.1083,E1 4.582,E2 405.8524} C_DIS
LIN {X 90.0765,Y 101.0384,Z 182,A 50.0796,B 4.4676,C 0.103,E1 4.5756,E2 402.729} C_DIS
LIN {X 86.7249,Y 103.9295,Z 182,A 51.6749,B 4.4676,C 0.1027,E1 4.5723,E2 401.1676} C_DIS
LIN {X 84.1712,Y 106.0079,Z 182,A 53.1477,B 4.4676,C 0.0993,E1 4.5691,E2 399.685} C_DIS
LIN {X 81.0021,Y 108.4487,Z 182,A 54.9453,B 4.4678,C 0.0951,E1 4.565,E2 397.8745} C_DIS
LIN {X 77.3876,Y 111.0567,Z 182,A 56.7724,B 4.4678,C 0.0926,E1 4.5609,E2 396.0547} C_DIS
LIN {X 73.9137,Y 113.3987,Z 182,A 58.5277,B 4.4678,C 0.09,E1 4.5568,E2 394.3015} C_DIS
LIN {X 70.4826,Y 115.5628,Z 182,A 60.2118,B 4.4679,C 0.0877,E1 4.5528,E2 392.6215} C_DIS
LIN {X 66.8025,Y 117.7283,Z 182,A 62.0057,B 4.4679,C 0.0852,E1 4.5485,E2 390.8292} C_DIS
LIN {X 63.4771,Y 119.553,Z 182,A 63.5236,B 4.468,C 0.084,E1 4.5448,E2 389.3221} C_DIS
LIN {X 60.1475,Y 121.261,Z 182,A 65.0916,B 4.468,C 0.082,E1 4.5409,E2 387.7561} C_DIS
LIN {X 57.2714,Y 122.6464,Z 182,A 66.4397,B 4.468,C 0.0804,E1 4.5375,E2 386.4085} C_DIS
LIN {X 54.2964,Y 123.9927,Z 182,A 67.8268,B 4.468,C 0.0787,E1 4.5339,E2 385.021} C_DIS
LIN {X 50.7772,Y 125.4736,Z 182,A 69.3393,B 4.4681,C 0.0779,E1 4.53,E2 383.5213} C_DIS
LIN {X 47.8389,Y 126.6235,Z 182,A 70.676,B 4.4681,C 0.0765,E1 4.5266,E2 382.1847} C_DIS
LIN {X 44.6482,Y 127.7833,Z 182,A 72.0782,B 4.4681,C 0.0754,E1 4.5229,E2 380.7869} C_DIS
LIN {X 40.9074,Y 129.0294,Z 182,A 73.9004,B 4.4682,C 0.0723,E1 4.518,E2 378.9465} C_DIS
LIN {X 36.3829,Y 130.3772,Z 182,A 75.69,B 4.4682,C 0.0727,E1 4.5132,E2 377.1826} C_DIS
LIN {X 33.2029,Y 131.2232,Z 182,A 77.0777,B 4.4682,C 0.0717,E1 4.5095,E2 375.796} C_DIS
LIN {X 29.4264,Y 132.1234,Z 182,A 78.8475,B 4.4682,C 0.0693,E1 4.5046,E2 374.0113} C_DIS
LIN {X 25.5017,Y 132.9347,Z 182,A 80.3832,B 4.4682,C 0.0699,E1 4.5005,E2 372.4955} C_DIS
LIN {X 22.1696,Y 133.5309,Z 182,A 81.8865,B 4.4682,C 0.0684,E1 4.4963,E2 370.9842} C_DIS
LIN {X 17.6127,Y 134.208,Z 182,A 83.7686,B 4.4682,C 0.0682,E1 4.4911,E2 369.1109} C_DIS
LIN {X 10.5206,Y 134.951,Z 182,A 86.9219,B 4.4683,C 0.0658,E1 4.4823,E2 365.9426} C_DIS
LIN {X 6.1421,Y 135.2211,Z 182,A 88.753,B 4.4683,C 0.0657,E1 4.4772,E2 364.1153} C_DIS
LIN {X -0.0619,Y 135.3596,Z 182,A 91.6882,B 4.4683,C 0.0625,E1 4.4689,E2 361.1438} C_DIS
LIN {X -4.1123,Y 135.2969,Z 182,A 93.0614,B 4.4683,C 0.0657,E1 4.4652,E2 359.8128} C_DIS
LIN {X -8.3852,Y 135.0989,Z 182,A 94.8238,B 4.4683,C 0.0663,E1 4.4603,E2 358.0571} C_DIS
LIN {X -13.268,Y 134.7074,Z 182,A 97.1858,B 4.4683,C 0.0641,E1 4.4536,E2 355.6611} C_DIS
LIN {X -16.8524,Y 134.3076,Z 182,A 98.4426,B 4.4683,C 0.067,E1 4.4503,E2 354.4379} C_DIS
LIN {X -20.4268,Y 133.8089,Z 182,A 99.9462,B 4.4683,C 0.0677,E1 4.4461,E2 352.9379} C_DIS
LIN {X -23.9497,Y 133.2231,Z 182,A 101.4609,B 4.4683,C 0.0683,E1 4.4419,E2 351.4237} C_DIS
LIN {X -27.9455,Y 132.444,Z 182,A 103.2073,B 4.4683,C 0.069,E1 4.4371,E2 349.6756} C_DIS
LIN {X -31.3212,Y 131.6856,Z 182,A 104.6372,B 4.4683,C 0.0701,E1 4.4333,E2 348.2506} C_DIS
LIN {X -34.5652,Y 130.8713,Z 182,A 106.1122,B 4.4683,C 0.0705,E1 4.4293,E2 346.7693} C_DIS
LIN {X -37.7855,Y 129.9779,Z 182,A 107.3582,B 4.4682,C 0.073,E1 4.426,E2 345.5444} C_DIS
LIN {X -41.238,Y 128.9238,Z 182,A 109.0245,B 4.4682,C 0.073,E1 4.4215,E2 343.8624} C_DIS
LIN {X -45.5269,Y 127.473,Z 182,A 111.4893,B 4.4682,C 0.07,E1 4.4148,E2 341.3325} C_DIS
LIN {X -49.7509,Y 125.8862,Z 182,A 112.9661,B 4.4682,C 0.0756,E1 4.4111,E2 339.9096} C_DIS
LIN {X -54.7062,Y 123.8123,Z 182,A 115.1951,B 4.4682,C 0.0783,E1 4.4054,E2 337.6875} C_DIS
LIN {X -58.1108,Y 122.2501,Z 182,A 116.7924,B 4.4681,C 0.08,E1 4.4014,E2 336.0899} C_DIS
LIN {X -61.0943,Y 120.787,Z 182,A 118.0452,B 4.4681,C 0.083,E1 4.3983,E2 334.8566} C_DIS
LIN {X -63.7311,Y 119.4191,Z 182,A 119.7593,B 4.4681,C 0.0809,E1 4.3939,E2 333.0882} C_DIS
LIN {X -68.1985,Y 116.9255,Z 182,A 121.5464,B 4.4679,C 0.0869,E1 4.3897,E2 331.3485} C_DIS
LIN {X -73.1113,Y 113.9174,Z 182,A 124.3395,B 4.4679,C 0.0876,E1 4.383,E2 328.5144} C_DIS
LIN {X -76.8259,Y 111.4463,Z 182,A 126.2165,B 4.4679,C 0.0907,E1 4.3786,E2 326.6403} C_DIS
LIN {X -80.4929,Y 108.8279,Z 182,A 128.1898,B 4.4679,C 0.0933,E1 4.3741,E2 324.6604} C_DIS
LIN {X -83.8906,Y 106.2305,Z 182,A 130.0153,B 4.4678,C 0.0962,E1 4.3701,E2 322.8344} C_DIS
LIN {X -87.2192,Y 103.5148,Z 182,A 131.87,B 4.4677,C 0.0992,E1 4.3661,E2 320.9767} C_DIS
LIN {X -90.4969,Y 100.6618,Z 182,A 133.6785,B 4.4677,C 0.1028,E1 4.3624,E2 319.1735} C_DIS
LIN {X -93.5889,Y 97.7934,Z 182,A 135.5588,B 4.4675,C 0.1055,E1 4.3585,E2 317.283} C_DIS
LIN {X -96.8684,Y 94.5466,Z 182,A 137.5593,B 4.4675,C 0.1091,E1 4.3546,E2 315.2784} C_DIS
LIN {X -99.8243,Y 91.4199,Z 182,A 139.4279,B 4.4674,C 0.1125,E1 4.351,E2 313.4055} C_DIS
LIN {X -102.7352,Y 88.1362,Z 182,A 141.3452,B 4.4673,C 0.116,E1 4.3475,E2 311.4824} C_DIS
LIN {X -105.6629,Y 84.6045,Z 182,A 143.3562,B 4.4672,C 0.1197,E1 4.3439,E2 309.4645} C_DIS
LIN {X -108.1704,Y 81.3735,Z 182,A 145.0961,B 4.4671,C 0.1235,E1 4.341,E2 307.725} C_DIS
LIN {X -110.8535,Y 77.6795,Z 182,A 147.1037,B 4.467,C 0.1274,E1 4.3377,E2 305.7098} C_DIS
LIN {X -112.8559,Y 74.7402,Z 182,A 148.6211,B 4.4669,C 0.1309,E1 4.3353,E2 304.1923} C_DIS
LIN {X -115.7333,Y 70.2016,Z 182,A 151.1072,B 4.4668,C 0.1349,E1 4.3317,E2 301.6821} C_DIS
LIN {X -118.2782,Y 65.8239,Z 182,A 153.1963,B 4.4666,C 0.1405,E1 4.3288,E2 299.6015} C_DIS
LIN {X -121.7839,Y 59.0866,Z 182,A 156.4774,B 4.4663,C 0.1482,E1 4.3246,E2 296.315} C_DIS
LIN {X -123.4929,Y 55.4205,Z 182,A 158.0987,B 4.4662,C 0.1532,E1 4.3227,E2 294.7062} C_DIS
LIN {X -124.8041,Y 52.4014,Z 182,A 159.5904,B 4.4661,C 0.1561,E1 4.3211,E2 293.2035} C_DIS
LIN {X -125.928,Y 49.6432,Z 182,A 160.9417,B 4.466,C 0.1589,E1 4.3197,E2 291.8422} C_DIS
LIN {X -127.0127,Y 46.7997,Z 182,A 162.7579,B 4.466,C 0.1588,E1 4.3179,E2 289.9619} C_DIS
LIN {X -128.4513,Y 42.687,Z 182,A 164.1133,B 4.4657,C 0.167,E1 4.3167,E2 288.6684} C_DIS
LIN {X -129.3357,Y 39.929,Z 182,A 165.4245,B 4.4656,C 0.1697,E1 4.3156,E2 287.3477} C_DIS
LIN {X -130.3753,Y 36.3898,Z 182,A 167.216,B 4.4655,C 0.1725,E1 4.3142,E2 285.529} C_DIS
LIN {X -131.66,Y 31.4274,Z 182,A 169.3181,B 4.4652,C 0.1789,E1 4.3128,E2 283.437} C_DIS
LIN {X -132.5235,Y 27.5648,Z 182,A 171.0065,B 4.465,C 0.1835,E1 4.3118,E2 281.7483} C_DIS
LIN {X -133.2081,Y 24.0335,Z 182,A 172.5172,B 4.4649,C 0.1878,E1 4.3111,E2 280.2402} C_DIS
LIN {X -133.7457,Y 20.8346,Z 182,A 174.0174,B 4.4647,C 0.1908,E1 4.3104,E2 278.7254} C_DIS
LIN {X -134.3437,Y 16.5544,Z 182,A 175.856,B 4.4645,C 0.1959,E1 4.3097,E2 276.8871} C_DIS
LIN {X -134.7399,Y 12.9292,Z 182,A 177.4721,B 4.4643,C 0.1998,E1 4.3092,E2 275.2631} C_DIS
LIN {X -135.0685,Y 8.8792,Z 182,A 179.3135,B 4.4641,C 0.2038,E1 4.3089,E2 273.408} C_DIS
LIN {X -135.2688,Y 4.9481,Z 182,A -179.0259,B 4.4639,C 0.2086,E1 4.3087,E2 271.7493} C_DIS
LIN {X -135.3576,Y 0.7679,Z 182,A -177.2111,B 4.4637,C 0.2133,E1 4.3086,E2 269.9301} C_DIS
LIN {X -135.3175,Y -3.3707,Z 182,A -175.3624,B 4.4635,C 0.2176,E1 4.3086,E2 268.0706} C_DIS
LIN {X -135.1827,Y -6.9046,Z 182,A -173.8237,B 4.4633,C 0.2216,E1 4.3089,E2 266.5277} C_DIS
LIN {X -134.8925,Y -11.2268,Z 182,A -172.0224,B 4.463,C 0.227,E1 4.3093,E2 264.7317} C_DIS
LIN {X -134.5709,Y -14.5835,Z 182,A -170.4563,B 4.4629,C 0.2301,E1 4.3097,E2 263.1492} C_DIS
LIN {X -134.0505,Y -18.7777,Z 182,A -168.5684,B 4.4626,C 0.2344,E1 4.3104,E2 261.25} C_DIS
LIN {X -133.4177,Y -22.8479,Z 182,A -166.8413,B 4.4624,C 0.2394,E1 4.3112,E2 259.5261} C_DIS
LIN {X -132.6892,Y -26.7509,Z 182,A -165.0658,B 4.4622,C 0.2434,E1 4.3121,E2 257.7397} C_DIS
LIN {X -131.9336,Y -30.2571,Z 182,A -163.5381,B 4.4619,C 0.2476,E1 4.313,E2 256.2118} C_DIS
LIN {X -131.016,Y -34.0194,Z 182,A -161.1915,B 4.4619,C 0.2472,E1 4.3148,E2 253.7767} C_DIS
LIN {X -129.6455,Y -38.9165,Z 182,A -159.5036,B 4.4615,C 0.2562,E1 4.316,E2 252.149} C_DIS
LIN {X -128.4574,Y -42.6688,Z 182,A -157.8647,B 4.4612,C 0.2609,E1 4.3174,E2 250.5144} C_DIS
LIN {X -126.1837,Y -48.9856,Z 182,A -154.9191,B 4.4608,C 0.2676,E1 4.3203,E2 247.5571} C_DIS
LIN {X -124.5445,Y -53.0203,Z 182,A -153.033,B 4.4605,C 0.2721,E1 4.3223,E2 245.6666} C_DIS
LIN {X -123.0412,Y -56.4175,Z 182,A -151.4216,B 4.4603,C 0.2758,E1 4.3242,E2 244.051} C_DIS
LIN {X -121.3098,Y -60.0487,Z 182,A -149.7316,B 4.46,C 0.2802,E1 4.3262,E2 242.3633} C_DIS
LIN {X -119.8793,Y -62.8557,Z 182,A -147.8315,B 4.46,C 0.2795,E1 4.3288,E2 240.3917} C_DIS
LIN {X -117.7772,Y -66.7146,Z 182,A -146.1902,B 4.4597,C 0.2856,E1 4.331,E2 238.7792} C_DIS
LIN {X -115.162,Y -71.136,Z 182,A -144.0684,B 4.4593,C 0.2911,E1 4.3341,E2 236.6649} C_DIS
LIN {X -112.9844,Y -74.5451,Z 182,A -142.3951,B 4.459,C 0.2954,E1 4.3366,E2 234.9971} C_DIS
LIN {X -110.6659,Y -77.9454,Z 182,A -140.5627,B 4.4588,C 0.2987,E1 4.3395,E2 233.1539} C_DIS
LIN {X -108.11,Y -81.4535,Z 182,A -138.6582,B 4.4586,C 0.3023,E1 4.3427,E2 231.2413} C_DIS
LIN {X -105.4225,Y -84.9031,Z 182,A -136.7539,B 4.4583,C 0.3058,E1 4.346,E2 229.3307} C_DIS
LIN {X -102.4658,Y -88.4489,Z 182,A -134.8185,B 4.458,C 0.3101,E1 4.3495,E2 227.3982} C_DIS
LIN {X -98.878,Y -92.4426,Z 182,A -132.4201,B 4.4578,C 0.3137,E1 4.3541,E2 224.9842} C_DIS
LIN {X -95.7928,Y -95.6361,Z 182,A -130.5481,B 4.4575,C 0.3174,E1 4.3577,E2 223.1135} C_DIS
LIN {X -92.6008,Y -98.7303,Z 182,A -128.566,B 4.4573,C 0.3202,E1 4.3618,E2 221.1189} C_DIS
LIN {X -89.2804,Y -101.7427,Z 182,A -126.5415,B 4.4572,C 0.3226,E1 4.366,E2 219.0784} C_DIS
LIN {X -85.5212,Y -104.9218,Z 182,A -124.5284,B 4.4569,C 0.3267,E1 4.3703,E2 217.0746} C_DIS
LIN {X -82.0005,Y -107.696,Z 182,A -122.5878,B 4.4567,C 0.3295,E1 4.3746,E2 215.1286} C_DIS
LIN {X -78.3524,Y -110.3789,Z 182,A -120.6611,B 4.4564,C 0.3324,E1 4.379,E2 213.2007} C_DIS
LIN {X -75.0358,Y -112.6592,Z 182,A -118.9272,B 4.4563,C 0.3347,E1 4.383,E2 211.4629} C_DIS
LIN {X -71.3693,Y -115.0169,Z 182,A -117.0217,B 4.4561,C 0.3368,E1 4.3875,E2 209.5496} C_DIS
LIN {X -67.4243,Y -117.3736,Z 182,A -115.0163,B 4.456,C 0.3388,E1 4.3924,E2 207.5364} C_DIS
LIN {X -63.5477,Y -119.5159,Z 182,A -113.1428,B 4.4558,C 0.3412,E1 4.397,E2 205.6628} C_DIS
LIN {X -60.2942,Y -121.1887,Z 182,A -111.6346,B 4.4556,C 0.3433,E1 4.4007,E2 204.1598} C_DIS
LIN {X -57.2436,Y -122.6592,Z 182,A -110.1796,B 4.4556,C 0.3447,E1 4.4044,E2 202.7018} C_DIS
LIN {X -53.8647,Y -124.1794,Z 182,A -108.6848,B 4.4553,C 0.347,E1 4.4082,E2 201.2163} C_DIS
LIN {X -50.8328,Y -125.4511,Z 182,A -107.2936,B 4.4553,C 0.3483,E1 4.4118,E2 199.8249} C_DIS
LIN {X -47.6888,Y -126.6796,Z 182,A -105.7761,B 4.4552,C 0.3488,E1 4.4158,E2 198.2957} C_DIS
LIN {X -44.1696,Y -127.9492,Z 182,A -103.9853,B 4.4552,C 0.3482,E1 4.4206,E2 196.4777} C_DIS
LIN {X -39.5595,Y -129.4487,Z 182,A -102.1238,B 4.455,C 0.3514,E1 4.4255,E2 194.6405} C_DIS
LIN {X -36.5694,Y -130.3251,Z 182,A -100.9032,B 4.4548,C 0.3532,E1 4.4287,E2 193.4322} C_DIS
LIN {X -33.8564,Y -131.0573,Z 182,A -99.4986,B 4.4549,C 0.3519,E1 4.4326,E2 191.9996} C_DIS
LIN {X -30.1778,Y -131.9517,Z 182,A -98.0187,B 4.4548,C 0.3539,E1 4.4366,E2 190.535} C_DIS
LIN {X -27.099,Y -132.6183,Z 182,A -96.7378,B 4.4547,C 0.355,E1 4.4401,E2 189.2605} C_DIS
LIN {X -23.9126,Y -133.2298,Z 182,A -95.2565,B 4.4547,C 0.3545,E1 4.4442,E2 187.7647} C_DIS
LIN {X -20.8333,Y -133.7459,Z 182,A -93.9318,B 4.4547,C 0.3549,E1 4.4478,E2 186.4392} C_DIS
LIN {X -13.4602,Y -134.6889,Z 182,A -90.6997,B 4.4547,C 0.3547,E1 4.4568,E2 183.195} C_DIS
LIN {X -9.3541,Y -135.0362,Z 182,A -89.0617,B 4.4547,C 0.3559,E1 4.4614,E2 181.5701} C_DIS
LIN {X -6.062,Y -135.2251,Z 182,A -87.5208,B 4.4547,C 0.3544,E1 4.4657,E2 180.0097} C_DIS
LIN {X 0.9561,Y -135.3453,Z 182,A -85.8027,B 4.4537,C 0.3669,E1 4.4702,E2 178.4515} C_DIS
Enddeposition()
LIN {X 0.9561,Y -135.3453,Z 182,A -85.8031,B 4.4537,C 0.3669,E1 4.4702,E2 178.4519} C_DIS
Startdeposition()
$VEL.CP = VEL_PRINT
LIN {X -1.4817,Y -136.2543,Z 182,A -86.7019,B 4.4082,C 0.3671,E1 4.4221,E2 179.381} C_DIS
LIN {X -5.3564,Y -136.1551,Z 182,A -87.6122,B 4.4088,C 0.36,E1 4.4198,E2 180.1991} C_DIS
LIN {X -7.9916,Y -136.0263,Z 182,A -89.2669,B 4.4084,C 0.3654,E1 4.415,E2 181.9249} C_DIS
LIN {X -12.5384,Y -135.683,Z 182,A -91.2231,B 4.4084,C 0.3656,E1 4.4095,E2 183.8869} C_DIS
LIN {X -15.7643,Y -135.3458,Z 182,A -92.7183,B 4.4083,C 0.3666,E1 4.4053,E2 185.3995} C_DIS
LIN {X -19.6982,Y -134.8296,Z 182,A -93.9571,B 4.4086,C 0.362,E1 4.4021,E2 186.5836} C_DIS
LIN {X -22.1467,Y -134.4486,Z 182,A -95.091,B 4.4086,C 0.3625,E1 4.3989,E2 187.7297} C_DIS
LIN {X -25.7171,Y -133.8113,Z 182,A -96.5552,B 4.4086,C 0.3614,E1 4.3949,E2 189.1866} C_DIS
LIN {X -29.1594,Y -133.1041,Z 182,A -98.127,B 4.4086,C 0.3616,E1 4.3906,E2 190.771} C_DIS
LIN {X -33.3646,Y -132.1122,Z 182,A -99.899,B 4.4088,C 0.3602,E1 4.3858,E2 192.5378} C_DIS
LIN {X -37.0429,Y -131.1287,Z 182,A -101.4597,B 4.4088,C 0.3588,E1 4.3816,E2 194.0937} C_DIS
LIN {X -40.6918,Y -130.0447,Z 182,A -103.343,B 4.4088,C 0.3603,E1 4.3765,E2 196.0138} C_DIS
LIN {X -44.9084,Y -128.6471,Z 182,A -104.9662,B 4.4091,C 0.3566,E1 4.3722,E2 197.6059} C_DIS
LIN {X -48.1237,Y -127.4794,Z 182,A -106.405,B 4.4091,C 0.3554,E1 4.3685,E2 199.0449} C_DIS
LIN {X -51.2503,Y -126.2548,Z 182,A -107.8718,B 4.4092,C 0.3546,E1 4.3646,E2 200.5191} C_DIS
LIN {X -54.3236,Y -124.9631,Z 182,A -109.2615,B 4.4094,C 0.3531,E1 4.3611,E2 201.9074} C_DIS
LIN {X -57.2139,Y -123.6661,Z 182,A -110.5957,B 4.4094,C 0.3517,E1 4.3577,E2 203.242} C_DIS
LIN {X -60.0606,Y -122.3091,Z 182,A -111.9874,B 4.4095,C 0.3508,E1 4.3542,E2 204.6424} C_DIS
LIN {X -63.301,Y -120.6637,Z 182,A -113.4838,B 4.4097,C 0.3487,E1 4.3505,E2 206.1348} C_DIS
LIN {X -66.8564,Y -118.733,Z 182,A -115.3318,B 4.4097,C 0.3478,E1 4.3459,E2 208.0018} C_DIS
LIN {X -70.7586,Y -116.45,Z 182,A -117.2862,B 4.4099,C 0.3457,E1 4.3412,E2 209.9632} C_DIS
LIN {X -74.3354,Y -114.1996,Z 182,A -119.093,B 4.4101,C 0.3434,E1 4.3369,E2 211.7738} C_DIS
LIN {X -78.1812,Y -111.6028,Z 182,A -121.0727,B 4.4103,C 0.3407,E1 4.3324,E2 213.7571} C_DIS
LIN {X -81.7124,Y -109.0438,Z 182,A -122.9535,B 4.4105,C 0.3382,E1 4.3281,E2 215.6438} C_DIS
LIN {X -85.2605,Y -106.2924,Z 182,A -124.8922,B 4.4107,C 0.3354,E1 4.3238,E2 217.5889} C_DIS
LIN {X -88.8198,Y -103.3361,Z 182,A -126.6208,B 4.4111,C 0.3303,E1 4.3202,E2 219.2895} C_DIS
LIN {X -91.2888,Y -101.1621,Z 182,A -128.2323,B 4.4111,C 0.3296,E1 4.3168,E2 220.9301} C_DIS
LIN {X -94.4897,Y -98.1792,Z 182,A -130.1525,B 4.4114,C 0.3268,E1 4.3129,E2 222.8602} C_DIS
LIN {X -97.0211,Y -95.6783,Z 182,A -131.6919,B 4.4116,C 0.3243,E1 4.3098,E2 224.4048} C_DIS
LIN {X -100.7609,Y -91.7309,Z 182,A -133.9473,B 4.4119,C 0.3195,E1 4.3055,E2 226.6558} C_DIS
LIN {X -103.1924,Y -88.9866,Z 182,A -135.5892,B 4.4121,C 0.317,E1 4.3025,E2 228.3101} C_DIS
LIN {X -106.1796,Y -85.4003,Z 182,A -137.5849,B 4.4124,C 0.3131,E1 4.299,E2 230.3095} C_DIS
LIN {X -108.9922,Y -81.781,Z 182,A -139.5722,B 4.4126,C 0.3093,E1 4.2956,E2 232.3038} C_DIS
LIN {X -111.6175,Y -78.1601,Z 182,A -141.5473,B 4.4129,C 0.3058,E1 4.2924,E2 234.2903} C_DIS
LIN {X -114.2387,Y -74.2753,Z 182,A -143.4653,B 4.4132,C 0.3008,E1 4.2894,E2 236.201} C_DIS
LIN {X -116.2831,Y -71.0324,Z 182,A -145.1985,B 4.4134,C 0.2979,E1 4.2868,E2 237.949} C_DIS
LIN {X -119.7842,Y -64.9551,Z 182,A -148.2142,B 4.4139,C 0.2912,E1 4.2827,E2 240.9719} C_DIS
LIN {X -121.5997,Y -61.4849,Z 182,A -149.8506,B 4.4141,C 0.2871,E1 4.2806,E2 242.6062} C_DIS
LIN {X -123.3812,Y -57.8302,Z 182,A -151.5188,B 4.4144,C 0.2825,E1 4.2786,E2 244.2684} C_DIS
LIN {X -124.6692,Y -54.9983,Z 182,A -152.9028,B 4.4146,C 0.2797,E1 4.277,E2 245.6614} C_DIS
LIN {X -125.7976,Y -52.3617,Z 182,A -154.1926,B 4.4148,C 0.2771,E1 4.2756,E2 246.9611} C_DIS
LIN {X -127.2676,Y -48.6853,Z 182,A -156.4663,B 4.4148,C 0.2769,E1 4.2732,E2 249.3104} C_DIS
LIN {X -128.846,Y -44.335,Z 182,A -157.9157,B 4.4153,C 0.2684,E1 4.2719,E2 250.6966} C_DIS
LIN {X -130.2777,Y -39.9313,Z 182,A -160.6247,B 4.4153,C 0.2682,E1 4.2696,E2 253.4997} C_DIS
LIN {X -131.7813,Y -34.6513,Z 182,A -162.2159,B 4.416,C 0.2572,E1 4.2685,E2 255.0001} C_DIS
LIN {X -132.5158,Y -31.724,Z 182,A -163.5819,B 4.4161,C 0.2544,E1 4.2676,E2 256.3775} C_DIS
LIN {X -133.2972,Y -28.2654,Z 182,A -165.2665,B 4.4163,C 0.2515,E1 4.2666,E2 258.0855} C_DIS
LIN {X -134.1212,Y -24.0485,Z 182,A -167.0054,B 4.4166,C 0.2461,E1 4.2657,E2 259.8148} C_DIS
LIN {X -134.7793,Y -20.0496,Z 182,A -168.9262,B 4.4168,C 0.2427,E1 4.2648,E2 261.7616} C_DIS
LIN {X -135.3055,Y -16.1023,Z 182,A -170.5131,B 4.4171,C 0.2375,E1 4.2643,E2 263.3364} C_DIS
LIN {X -135.7238,Y -12.0959,Z 182,A -172.3286,B 4.4173,C 0.2335,E1 4.2638,E2 265.166} C_DIS
LIN {X -136.0054,Y -8.332,Z 182,A -173.8943,B 4.4175,C 0.2289,E1 4.2635,E2 266.7279} C_DIS
LIN {X -136.1972,Y -4.166,Z 182,A -175.7573,B 4.4177,C 0.2246,E1 4.2633,E2 268.6033} C_DIS
LIN {X -136.2614,Y -0.3696,Z 182,A -177.4898,B 4.4179,C 0.221,E1 4.2633,E2 270.3516} C_DIS
LIN {X -136.1954,Y 4.2325,Z 182,A -179.3339,B 4.4182,C 0.2149,E1 4.2633,E2 272.183} C_DIS
LIN {X -136.0272,Y 7.978,Z 182,A 178.958,B 4.4184,C 0.2113,E1 4.2636,E2 273.9062} C_DIS
LIN {X -135.7716,Y 11.5303,Z 182,A 177.4724,B 4.4186,C 0.207,E1 4.2639,E2 275.3892} C_DIS
LIN {X -135.3746,Y 15.5228,Z 182,A 175.6197,B 4.4188,C 0.2033,E1 4.2645,E2 277.2611} C_DIS
LIN {X -134.8262,Y 19.7217,Z 182,A 173.9471,B 4.419,C 0.1976,E1 4.2651,E2 278.919} C_DIS
LIN {X -134.3673,Y 22.6343,Z 182,A 172.5578,B 4.4191,C 0.1951,E1 4.2657,E2 280.3258} C_DIS
LIN {X -133.6096,Y 26.7486,Z 182,A 170.7388,B 4.4193,C 0.1906,E1 4.2667,E2 282.1509} C_DIS
LIN {X -132.8254,Y 30.4011,Z 182,A 169.1607,B 4.4195,C 0.1862,E1 4.2677,E2 283.7286} C_DIS
LIN {X -131.9429,Y 34.0316,Z 182,A 167.0708,B 4.4195,C 0.1853,E1 4.2691,E2 285.8809} C_DIS
LIN {X -130.8619,Y 37.9743,Z 182,A 165.8217,B 4.4199,C 0.1776,E1 4.2701,E2 287.071} C_DIS
LIN {X -130.0622,Y 40.6355,Z 182,A 164.3171,B 4.4199,C 0.1766,E1 4.2713,E2 288.616} C_DIS
LIN {X -127.872,Y 47.0757,Z 182,A 161.641,B 4.4203,C 0.1677,E1 4.2738,E2 291.2672} C_DIS
LIN {X -126.8104,Y 49.8614,Z 182,A 160.3087,B 4.4203,C 0.1649,E1 4.2751,E2 292.6081} C_DIS
LIN {X -125.6168,Y 52.7945,Z 182,A 158.9229,B 4.4205,C 0.1618,E1 4.2766,E2 293.9994} C_DIS
LIN {X -124.2589,Y 55.9156,Z 182,A 157.4684,B 4.4206,C 0.1582,E1 4.2782,E2 295.4556} C_DIS
LIN {X -122.5755,Y 59.5205,Z 182,A 154.7937,B 4.4206,C 0.1606,E1 4.2817,E2 298.2504} C_DIS
LIN {X -119.5586,Y 65.3686,Z 182,A 152.9826,B 4.421,C 0.1474,E1 4.2839,E2 299.9435} C_DIS
LIN {X -116.0966,Y 71.3363,Z 182,A 149.3945,B 4.421,C 0.1449,E1 4.2891,E2 303.6127} C_DIS
LIN {X -113.7574,Y 75.0104,Z 182,A 148.051,B 4.4213,C 0.1373,E1 4.2911,E2 304.8956} C_DIS
LIN {X -111.8294,Y 77.8554,Z 182,A 146.4391,B 4.4213,C 0.1351,E1 4.2937,E2 306.5265} C_DIS
LIN {X -109.2393,Y 81.4499,Z 182,A 144.5356,B 4.4215,C 0.1311,E1 4.2968,E2 308.4334} C_DIS
LIN {X -106.4539,Y 85.0584,Z 182,A 142.5851,B 4.4216,C 0.1271,E1 4.3002,E2 310.3864} C_DIS
LIN {X -103.8152,Y 88.2592,Z 182,A 140.7773,B 4.4217,C 0.1238,E1 4.3034,E2 312.2005} C_DIS
LIN {X -100.8885,Y 91.5904,Z 182,A 138.8668,B 4.4218,C 0.1202,E1 4.307,E2 314.115} C_DIS
LIN {X -97.79,Y 94.8916,Z 182,A 136.9038,B 4.4219,C 0.1168,E1 4.3108,E2 316.0837} C_DIS
LIN {X -94.5747,Y 98.0969,Z 182,A 134.9595,B 4.4219,C 0.1133,E1 4.3147,E2 318.0307} C_DIS
LIN {X -91.3058,Y 101.1467,Z 182,A 133.0226,B 4.4221,C 0.1102,E1 4.3186,E2 319.9729} C_DIS
LIN {X -87.8867,Y 104.1315,Z 182,A 131.0465,B 4.4221,C 0.1072,E1 4.3229,E2 321.9557} C_DIS
LIN {X -84.3507,Y 107.0154,Z 182,A 129.107,B 4.4222,C 0.104,E1 4.3271,E2 323.8962} C_DIS
LIN {X -80.756,Y 109.7532,Z 182,A 127.2006,B 4.4222,C 0.1009,E1 4.3313,E2 325.8019} C_DIS
LIN {X -77.1666,Y 112.3059,Z 182,A 125.3157,B 4.4224,C 0.0982,E1 4.3357,E2 327.6894} C_DIS
LIN {X -70.2565,Y 116.7536,Z 182,A 121.9148,B 4.4224,C 0.0927,E1 4.3437,E2 331.0812} C_DIS
LIN {X -67.1191,Y 118.5854,Z 182,A 120.1848,B 4.4224,C 0.0922,E1 4.3479,E2 332.8345} C_DIS
LIN {X -63.3455,Y 120.6403,Z 182,A 118.3369,B 4.4225,C 0.0902,E1 4.3525,E2 334.6859} C_DIS
LIN {X -59.9951,Y 122.3414,Z 182,A 116.8832,B 4.4225,C 0.0873,E1 4.3561,E2 336.1233} C_DIS
LIN {X -56.5427,Y 123.9765,Z 182,A 115.2677,B 4.4226,C 0.0855,E1 4.3602,E2 337.7389} C_DIS
LIN {X -51.7937,Y 126.0348,Z 182,A 113.0684,B 4.4226,C 0.0834,E1 4.3658,E2 339.9396} C_DIS
LIN {X -48.6786,Y 127.2698,Z 182,A 110.875,B 4.4226,C 0.0885,E1 4.3718,E2 342.2257} C_DIS
LIN {X -43.3453,Y 129.1823,Z 182,A 109.4372,B 4.4227,C 0.0786,E1 4.3753,E2 343.5491} C_DIS
LIN {X -39.2974,Y 130.4717,Z 182,A 107.3185,B 4.4227,C 0.08,E1 4.381,E2 345.7067} C_DIS
LIN {X -34.6837,Y 131.7727,Z 182,A 105.3582,B 4.4227,C 0.0782,E1 4.3863,E2 347.6591} C_DIS
LIN {X -30.5658,Y 132.7878,Z 182,A 103.5811,B 4.4227,C 0.077,E1 4.3911,E2 349.4345} C_DIS
LIN {X -26.9693,Y 133.5647,Z 182,A 102.0334,B 4.4227,C 0.0762,E1 4.3953,E2 350.9813} C_DIS
LIN {X -23.077,Y 134.2934,Z 182,A 100.2864,B 4.4227,C 0.0762,E1 4.4002,E2 352.7373} C_DIS
LIN {X -19.0693,Y 134.9194,Z 182,A 98.6372,B 4.4228,C 0.0751,E1 4.4047,E2 354.3787} C_DIS
LIN {X -14.9133,Y 135.4421,Z 182,A 96.4484,B 4.4228,C 0.0785,E1 4.4109,E2 356.6178} C_DIS
LIN {X -10.7852,Y 135.8345,Z 182,A 95.2134,B 4.4228,C 0.0736,E1 4.4142,E2 357.7911} C_DIS
LIN {X -6.6305,Y 136.0991,Z 182,A 93.3628,B 4.4228,C 0.0744,E1 4.4194,E2 359.6529} C_DIS
LIN {X 1.3525,Y 136.255,Z 182,A 90.0699,B 4.4228,C 0.0739,E1 4.4286,E2 362.9366} C_DIS
LIN {X 6.1398,Y 136.1238,Z 182,A 87.9069,B 4.4228,C 0.0756,E1 4.4347,E2 365.1168} C_DIS
LIN {X 10.1875,Y 135.8792,Z 182,A 85.9114,B 4.4228,C 0.0788,E1 4.4403,E2 367.1463} C_DIS
LIN {X 14.0903,Y 135.5302,Z 182,A 84.6597,B 4.4228,C 0.0756,E1 4.4437,E2 368.35} C_DIS
LIN {X 17.8502,Y 135.086,Z 182,A 83.0647,B 4.4228,C 0.0763,E1 4.4481,E2 369.9449} C_DIS
LIN {X 21.2771,Y 134.5894,Z 182,A 81.6362,B 4.4228,C 0.0767,E1 4.452,E2 371.3696} C_DIS
LIN {X 25.3754,Y 133.8767,Z 182,A 79.9146,B 4.4228,C 0.0774,E1 4.4567,E2 373.0874} C_DIS
LIN {X 28.7351,Y 133.1958,Z 182,A 78.5011,B 4.4228,C 0.0781,E1 4.4606,E2 374.497} C_DIS
LIN {X 31.8902,Y 132.4758,Z 182,A 77.102,B 4.4228,C 0.0794,E1 4.4644,E2 375.9004} C_DIS
LIN {X 35.4004,Y 131.5815,Z 182,A 75.5834,B 4.4228,C 0.0806,E1 4.4685,E2 377.4181} C_DIS
LIN {X 40.3123,Y 130.1611,Z 182,A 73.4807,B 4.4227,C 0.082,E1 4.4741,E2 379.5146} C_DIS
LIN {X 43.3696,Y 129.1742,Z 182,A 72.1348,B 4.4227,C 0.0832,E1 4.4777,E2 380.8597} C_DIS
LIN {X 47.4581,Y 127.7287,Z 182,A 70.3162,B 4.4227,C 0.085,E1 4.4825,E2 382.6774} C_DIS
LIN {X 51.1476,Y 126.2962,Z 182,A 68.7718,B 4.4227,C 0.0855,E1 4.4864,E2 384.2071} C_DIS
LIN {X 54.3439,Y 124.9543,Z 182,A 67.2401,B 4.4226,C 0.088,E1 4.4904,E2 385.7476} C_DIS
LIN {X 57.5923,Y 123.4911,Z 182,A 65.8127,B 4.4226,C 0.0891,E1 4.494,E2 387.1662} C_DIS
LIN {X 60.6409,Y 122.0229,Z 182,A 64.4153,B 4.4226,C 0.0907,E1 4.4975,E2 388.5603} C_DIS
LIN {X 63.5425,Y 120.5368,Z 182,A 63.0455,B 4.4225,C 0.0925,E1 4.5009,E2 389.93} C_DIS
LIN {X 67.2031,Y 118.5376,Z 182,A 61.216,B 4.4225,C 0.0959,E1 4.5054,E2 391.7686} C_DIS
LIN {X 71.0122,Y 116.2955,Z 182,A 59.3742,B 4.4223,C 0.0985,E1 4.5098,E2 393.6084} C_DIS
LIN {X 74.9976,Y 113.7658,Z 182,A 57.4848,B 4.4223,C 0.1006,E1 4.5142,E2 395.4862} C_DIS
LIN {X 78.5016,Y 111.3768,Z 182,A 55.6978,B 4.4223,C 0.1035,E1 4.5183,E2 397.2737} C_DIS
LIN {X 82.2716,Y 108.622,Z 182,A 53.6028,B 4.4221,C 0.1084,E1 4.523,E2 399.3848} C_DIS
LIN {X 86.8467,Y 104.9997,Z 182,A 51.4774,B 4.4221,C 0.1091,E1 4.5276,E2 401.4706} C_DIS
LIN {X 89.8703,Y 102.4244,Z 182,A 49.7382,B 4.422,C 0.1131,E1 4.5313,E2 403.2185} C_DIS
LIN {X 95.5913,Y 97.1064,Z 182,A 46.6845,B 4.422,C 0.1169,E1 4.5374,E2 406.2445} C_DIS
LIN {X 99.6086,Y 92.9808,Z 182,A 44.2647,B 4.4218,C 0.1219,E1 4.5421,E2 408.6647} C_DIS
LIN {X 102.3024,Y 90.009,Z 182,A 42.5087,B 4.4216,C 0.1263,E1 4.5454,E2 410.4296} C_DIS
LIN {X 105.4519,Y 86.2971,Z 182,A 40.5967,B 4.4216,C 0.1292,E1 4.5488,E2 412.3256} C_DIS
LIN {X 108.117,Y 82.934,Z 182,A 38.9336,B 4.4215,C 0.1316,E1 4.5516,E2 413.9719} C_DIS
LIN {X 110.1444,Y 80.2223,Z 182,A 37.3371,B 4.4213,C 0.1369,E1 4.5543,E2 415.59} C_DIS
LIN {X 112.7818,Y 76.4695,Z 182,A 35.5242,B 4.4213,C 0.14,E1 4.5572,E2 417.3893} C_DIS
LIN {X 115.127,Y 72.891,Z 182,A 33.7354,B 4.4211,C 0.1442,E1 4.5599,E2 419.1775} C_DIS
LIN {X 117.5277,Y 68.9532,Z 182,A 31.8661,B 4.421,C 0.1481,E1 4.5626,E2 421.039} C_DIS
LIN {X 119.7985,Y 64.9288,Z 182,A 29.9478,B 4.4208,C 0.1526,E1 4.5652,E2 422.955} C_DIS
LIN {X 121.5724,Y 61.5384,Z 182,A 28.5026,B 4.4208,C 0.1547,E1 4.567,E2 424.3805} C_DIS
LIN {X 123.0162,Y 58.5984,Z 182,A 27.1301,B 4.4206,C 0.1582,E1 4.5686,E2 425.7531} C_DIS
LIN {X 124.7819,Y 54.7427,Z 182,A 24.8923,B 4.4202,C 0.1684,E1 4.5713,E2 428.0477} C_DIS
LIN {X 126.5544,Y 50.5071,Z 182,A 23.5455,B 4.4203,C 0.1662,E1 4.5726,E2 429.3235} C_DIS
LIN {X 127.686,Y 47.572,Z 182,A 22.2749,B 4.4203,C 0.1691,E1 4.5738,E2 430.5883} C_DIS
LIN {X 128.7587,Y 44.5868,Z 182,A 20.9541,B 4.4201,C 0.1725,E1 4.5751,E2 431.9082} C_DIS
LIN {X 129.8819,Y 41.2013,Z 182,A 19.5774,B 4.42,C 0.175,E1 4.5762,E2 433.2704} C_DIS
LIN {X 130.7085,Y 38.4982,Z 182,A 18.3153,B 4.4198,C 0.1792,E1 4.5773,E2 434.5423} C_DIS
LIN {X 131.7066,Y 34.9313,Z 182,A 16.8595,B 4.4197,C 0.1821,E1 4.5783,E2 435.9863} C_DIS
LIN {X 132.4772,Y 31.8842,Z 182,A 15.5579,B 4.4196,C 0.1855,E1 4.5792,E2 437.2861} C_DIS
LIN {X 133.3317,Y 28.1053,Z 182,A 14.0189,B 4.4194,C 0.1889,E1 4.5801,E2 438.8149} C_DIS
LIN {X 133.8743,Y 25.3877,Z 182,A 12.8398,B 4.4193,C 0.1923,E1 4.5807,E2 439.9965} C_DIS
LIN {X 134.5353,Y 21.6265,Z 182,A 11.2302,B 4.4191,C 0.1969,E1 4.5815,E2 441.6077} C_DIS
LIN {X 135.1958,Y 17.0128,Z 182,A 9.1743,B 4.4188,C 0.2036,E1 4.5822,E2 443.6767} C_DIS
LIN {X 135.7274,Y 12.0539,Z 182,A 7.3115,B 4.4186,C 0.2065,E1 4.5827,E2 445.5117} C_DIS
LIN {X 136.174,Y 4.872,Z 182,A 4.2133,B 4.4182,C 0.216,E1 4.5832,E2 448.6211} C_DIS
LIN {X 136.2519,Y -1.6433,Z 182,A 1.8817,B 4.4181,C 0.2186,E1 4.5832,E2 450.9034} C_DIS
LIN {X 135.9714,Y -8.8838,Z 182,A -1.5852,B 4.4173,C 0.2326,E1 4.5828,E2 454.4252} C_DIS
LIN {X 135.6469,Y -12.915,Z 182,A -2.7978,B 4.4174,C 0.2311,E1 4.5825,E2 455.5778} C_DIS
LIN {X 135.2826,Y -16.2937,Z 182,A -4.2016,B 4.4172,C 0.2349,E1 4.582,E2 456.9796} C_DIS
LIN {X 134.4349,Y -22.2291,Z 182,A -6.734,B 4.4168,C 0.2421,E1 4.581,E2 459.5153} C_DIS
LIN {X 133.6177,Y -26.7086,Z 182,A -8.5421,B 4.4166,C 0.2461,E1 4.58,E2 461.3116} C_DIS
LIN {X 132.847,Y -30.3064,Z 182,A -10.0236,B 4.4164,C 0.2495,E1 4.5791,E2 462.7859} C_DIS
LIN {X 132.0557,Y -33.587,Z 182,A -11.3546,B 4.4163,C 0.2523,E1 4.5783,E2 464.1069} C_DIS
LIN {X 131.1587,Y -36.9359,Z 182,A -12.7391,B 4.4161,C 0.2554,E1 4.5772,E2 465.4833} C_DIS
LIN {X 130.1511,Y -40.3449,Z 182,A -14.179,B 4.4159,C 0.2588,E1 4.5761,E2 466.9174} C_DIS
LIN {X 129.1033,Y -43.5824,Z 182,A -15.9131,B 4.4154,C 0.2665,E1 4.5745,E2 468.6912} C_DIS
LIN {X 127.9607,Y -46.8323,Z 182,A -16.9833,B 4.4154,C 0.2656,E1 4.5736,E2 469.7146} C_DIS
LIN {X 126.7346,Y -50.0562,Z 182,A -18.6695,B 4.4151,C 0.2725,E1 4.5718,E2 471.432} C_DIS
LIN {X 124.9386,Y -54.3803,Z 182,A -20.3384,B 4.415,C 0.2739,E1 4.57,E2 473.0644} C_DIS
LIN {X 123.6143,Y -57.3261,Z 182,A -21.7461,B 4.4147,C 0.2781,E1 4.5684,E2 474.4795} C_DIS
LIN {X 121.4624,Y -61.7545,Z 182,A -23.9282,B 4.4143,C 0.2848,E1 4.5656,E2 476.6776} C_DIS
LIN {X 119.8888,Y -64.7616,Z 182,A -25.0802,B 4.4143,C 0.285,E1 4.5642,E2 477.7958} C_DIS
LIN {X 117.761,Y -68.5547,Z 182,A -26.9222,B 4.414,C 0.2897,E1 4.5616,E2 479.6411} C_DIS
LIN {X 115.4169,Y -72.4318,Z 182,A -28.8042,B 4.4137,C 0.2941,E1 4.5589,E2 481.5218} C_DIS
LIN {X 112.8893,Y -76.3106,Z 182,A -30.6051,B 4.4135,C 0.297,E1 4.5561,E2 483.3058} C_DIS
LIN {X 110.5201,Y -79.7039,Z 182,A -32.3801,B 4.4132,C 0.3015,E1 4.5532,E2 485.0867} C_DIS
LIN {X 107.8429,Y -83.2902,Z 182,A -34.1935,B 4.4129,C 0.305,E1 4.5502,E2 486.8929} C_DIS
LIN {X 105.1099,Y -86.7137,Z 182,A -35.994,B 4.4127,C 0.3087,E1 4.547,E2 488.6896} C_DIS
LIN {X 101.4923,Y -90.9209,Z 182,A -38.5586,B 4.4121,C 0.3167,E1 4.5422,E2 491.2858} C_DIS
LIN {X 98.8466,Y -93.7912,Z 182,A -39.84,B 4.4121,C 0.3158,E1 4.5399,E2 492.5226} C_DIS
LIN {X 95.875,Y -96.8263,Z 182,A -42.0911,B 4.4115,C 0.3251,E1 4.5353,E2 494.8346} C_DIS
LIN {X 92.3567,Y -100.1872,Z 182,A -43.5822,B 4.4117,C 0.3225,E1 4.5324,E2 496.2564} C_DIS
LIN {X 89.5458,Y -102.7075,Z 182,A -45.0069,B 4.4117,C 0.3237,E1 4.5294,E2 497.6615} C_DIS
LIN {X 86.6556,Y -105.158,Z 182,A -46.6773,B 4.4113,C 0.3277,E1 4.5258,E2 499.3431} C_DIS
LIN {X 83.3578,Y -107.7904,Z 182,A -48.5888,B 4.4109,C 0.3326,E1 4.5216,E2 501.2737} C_DIS
LIN {X 79.3769,Y -110.7548,Z 182,A -50.5242,B 4.4109,C 0.3344,E1 4.5173,E2 503.1913} C_DIS
LIN {X 75.8691,Y -113.1867,Z 182,A -52.1958,B 4.4107,C 0.336,E1 4.5134,E2 504.8485} C_DIS
LIN {X 72.5452,Y -115.3453,Z 182,A -53.8458,B 4.4105,C 0.3386,E1 4.5096,E2 506.4977} C_DIS
LIN {X 68.9848,Y -117.5091,Z 182,A -55.6213,B 4.4103,C 0.3416,E1 4.5053,E2 508.2775} C_DIS
LIN {X 64.9316,Y -119.797,Z 182,A -57.5667,B 4.41,C 0.3443,E1 4.5005,E2 510.2229} C_DIS
LIN {X 61.7188,Y -121.4806,Z 182,A -58.9518,B 4.41,C 0.3449,E1 4.4971,E2 511.591} C_DIS
LIN {X 57.7639,Y -123.4118,Z 182,A -60.7545,B 4.4099,C 0.3468,E1 4.4926,E2 513.3889} C_DIS
LIN {X 54.6763,Y -124.8106,Z 182,A -62.373,B 4.4095,C 0.3508,E1 4.4884,E2 515.0334} C_DIS
LIN {X 46.4627,Y -128.0939,Z 182,A -65.7686,B 4.4095,C 0.3515,E1 4.4797,E2 518.3897} C_DIS
LIN {X 42.7259,Y -129.3885,Z 182,A -67.4525,B 4.4093,C 0.3534,E1 4.4752,E2 520.0775} C_DIS
LIN {X 39.6137,Y -130.3749,Z 182,A -68.8102,B 4.4093,C 0.3546,E1 4.4716,E2 521.4342} C_DIS
LIN {X 36.702,Y -131.2241,Z 182,A -70.1212,B 4.4091,C 0.3561,E1 4.4681,E2 522.7506} C_DIS
LIN {X 33.5873,Y -132.0557,Z 182,A -71.4518,B 4.4091,C 0.357,E1 4.4645,E2 524.0788} C_DIS
LIN {X 30.3064,Y -132.847,Z 182,A -72.8556,B 4.409,C 0.3579,E1 4.4607,E2 525.4815} C_DIS
LIN {X 26.9801,Y -133.5625,Z 182,A -74.2949,B 4.4089,C 0.359,E1 4.4567,E2 526.9228} C_DIS
LIN {X 20.6186,Y -134.6914,Z 182,A -77.2389,B 4.4085,C 0.3631,E1 4.4485,E2 529.8978} C_DIS
LIN {X 15.4841,Y -135.3792,Z 182,A -79.9251,B 4.408,C 0.3694,E1 4.4409,E2 532.6505} C_DIS
LIN {X 9.6481,Y -135.9186,Z 182,A -81.5074,B 4.4087,C 0.3612,E1 4.4368,E2 534.1205} C_DIS
LIN {X 2.0663,Y -136.2449,Z 182,A -84.7308,B 4.4087,C 0.3623,E1 4.4278,E2 537.3498} C_DIS
LIN {X 2.0663,Y -136.2449,Z 182,A -84.7308,B 4.4087,C 0.3623,E1 4.4278,E2 537.3498} C_DIS
Enddeposition()
LIN {X 0.9727,Y -137.1551,Z 182,A -84.8196,B 4.3967,C 0.3608,E1 4.4155,E2 537.4255} C_DIS
Startdeposition()
$VEL.CP = VEL_PRINT
LIN {X 5.6935,Y -137.0441,Z 182,A -82.2822,B 4.3972,C 0.3545,E1 4.4228,E2 534.8128} C_DIS
LIN {X 9.267,Y -136.8503,Z 182,A -80.9414,B 4.3971,C 0.3556,E1 4.4265,E2 533.4917} C_DIS
LIN {X 13.3751,Y -136.5083,Z 182,A -79.4006,B 4.397,C 0.3569,E1 4.4307,E2 531.9739} C_DIS
LIN {X 17.5306,Y -136.0371,Z 182,A -76.7243,B 4.3979,C 0.346,E1 4.4385,E2 529.173} C_DIS
LIN {X 24.2788,Y -134.9958,Z 182,A -74.8508,B 4.3972,C 0.3549,E1 4.4433,E2 527.4281} C_DIS
LIN {X 27.5392,Y -134.3686,Z 182,A -73.4657,B 4.3972,C 0.354,E1 4.4471,E2 526.0424} C_DIS
LIN {X 30.7114,Y -133.6792,Z 182,A -72.1061,B 4.3973,C 0.3529,E1 4.4508,E2 524.6815} C_DIS
LIN {X 34.074,Y -132.8622,Z 182,A -70.6955,B 4.3973,C 0.3521,E1 4.4546,E2 523.2746} C_DIS
LIN {X 37.6016,Y -131.9086,Z 182,A -69.1876,B 4.3975,C 0.351,E1 4.4587,E2 521.7682} C_DIS
LIN {X 40.4072,Y -131.0748,Z 182,A -67.9414,B 4.3975,C 0.3496,E1 4.462,E2 520.5181} C_DIS
LIN {X 44.198,Y -129.8464,Z 182,A -66.2118,B 4.3978,C 0.3471,E1 4.4666,E2 518.7788} C_DIS
LIN {X 52.6153,Y -126.6686,Z 182,A -62.8166,B 4.3978,C 0.3471,E1 4.4754,E2 515.429} C_DIS
LIN {X 58.5116,Y -124.0567,Z 182,A -60.0095,B 4.3982,C 0.3423,E1 4.4826,E2 512.6052} C_DIS
LIN {X 62.6307,Y -122.0279,Z 182,A -57.9977,B 4.3984,C 0.3386,E1 4.4876,E2 510.5796} C_DIS
LIN {X 65.9503,Y -120.2682,Z 182,A -56.4096,B 4.3986,C 0.3361,E1 4.4916,E2 508.9879} C_DIS
LIN {X 69.9205,Y -118.0044,Z 182,A -54.5894,B 4.3988,C 0.3342,E1 4.4959,E2 507.178} C_DIS
LIN {X 73.554,Y -115.7746,Z 182,A -52.7822,B 4.399,C 0.331,E1 4.5002,E2 505.3659} C_DIS
LIN {X 77.222,Y -113.3609,Z 182,A -50.9935,B 4.3992,C 0.3285,E1 4.5044,E2 503.5817} C_DIS
LIN {X 81.0983,Y -110.6203,Z 182,A -49.1113,B 4.3994,C 0.3262,E1 4.5086,E2 501.7112} C_DIS
LIN {X 83.5811,Y -108.7569,Z 182,A -47.8608,B 4.3995,C 0.3244,E1 4.5114,E2 500.4658} C_DIS
LIN {X 86.6383,Y -106.3373,Z 182,A -46.1707,B 4.3998,C 0.3207,E1 4.5151,E2 498.7663} C_DIS
LIN {X 91.9941,Y -101.7394,Z 182,A -42.7649,B 4.4006,C 0.3093,E1 4.5223,E2 495.2977} C_DIS
LIN {X 95.7973,Y -98.1666,Z 182,A -41.2414,B 4.4003,C 0.3129,E1 4.5252,E2 493.8589} C_DIS
LIN {X 98.7784,Y -95.1666,Z 182,A -38.4683,B 4.4015,C 0.2967,E1 4.5309,E2 490.9513} C_DIS
LIN {X 103.9446,Y -89.4947,Z 182,A -36.5258,B 4.4009,C 0.3055,E1 4.5341,E2 489.1728} C_DIS
LIN {X 106.1302,Y -86.8917,Z 182,A -34.9379,B 4.4012,C 0.3002,E1 4.537,E2 487.5618} C_DIS
LIN {X 108.875,Y -83.4268,Z 182,A -33.1545,B 4.4015,C 0.2967,E1 4.54,E2 485.785} C_DIS
LIN {X 111.4417,Y -79.966,Z 182,A -31.4356,B 4.4017,C 0.2935,E1 4.5429,E2 484.0752} C_DIS
LIN {X 113.7741,Y -76.6116,Z 182,A -29.6986,B 4.402,C 0.289,E1 4.5456,E2 482.3328} C_DIS
LIN {X 116.2644,Y -72.777,Z 182,A -27.8556,B 4.4022,C 0.2852,E1 4.5484,E2 480.4969} C_DIS
LIN {X 118.521,Y -69.0412,Z 182,A -26.1174,B 4.4024,C 0.2818,E1 4.5508,E2 478.7683} C_DIS
LIN {X 120.6413,Y -65.2656,Z 182,A -24.0075,B 4.403,C 0.2734,E1 4.5537,E2 476.6175} C_DIS
LIN {X 122.4612,Y -61.7792,Z 182,A -22.7683,B 4.403,C 0.2743,E1 4.5552,E2 475.4296} C_DIS
LIN {X 124.6817,Y -57.1654,Z 182,A -20.7831,B 4.4031,C 0.2708,E1 4.5576,E2 473.4626} C_DIS
LIN {X 125.8432,Y -54.5594,Z 182,A -19.5832,B 4.4033,C 0.2675,E1 4.5589,E2 472.2605} C_DIS
LIN {X 127.3335,Y -50.9854,Z 182,A -17.9653,B 4.4036,C 0.2632,E1 4.5606,E2 470.6412} C_DIS
LIN {X 128.8554,Y -47.0087,Z 182,A -16.1402,B 4.4039,C 0.2579,E1 4.5624,E2 468.8087} C_DIS
LIN {X 130.3839,Y -42.5902,Z 182,A -14.4238,B 4.404,C 0.2556,E1 4.5639,E2 467.1214} C_DIS
LIN {X 131.313,Y -39.6287,Z 182,A -13.1857,B 4.4042,C 0.2528,E1 4.5649,E2 465.8898} C_DIS
LIN {X 132.0677,Y -37.0325,Z 182,A -11.972,B 4.4044,C 0.2486,E1 4.5658,E2 464.6643} C_DIS
LIN {X 132.9978,Y -33.5396,Z 182,A -10.5813,B 4.4046,C 0.246,E1 4.5668,E2 463.2877} C_DIS
LIN {X 133.9534,Y -29.4975,Z 182,A -8.84,B 4.4048,C 0.2411,E1 4.5679,E2 461.5443} C_DIS
LIN {X 134.7163,Y -25.7845,Z 182,A -6.4439,B 4.4056,C 0.2261,E1 4.5692,E2 459.0412} C_DIS
LIN {X 135.8555,Y -18.8915,Z 182,A -4.5694,B 4.4054,C 0.2315,E1 4.5699,E2 457.3001} C_DIS
LIN {X 136.3255,Y -15.1293,Z 182,A -2.4023,B 4.406,C 0.2194,E1 4.5706,E2 455.0565} C_DIS
LIN {X 136.7942,Y -10.0354,Z 182,A -0.9015,B 4.4059,C 0.2217,E1 4.5709,E2 453.6363} C_DIS
LIN {X 137.0327,Y -5.9849,Z 182,A 0.7769,B 4.4061,C 0.2171,E1 4.5711,E2 451.9588} C_DIS
LIN {X 137.1435,Y -2.2476,Z 182,A 2.8453,B 4.4066,C 0.2061,E1 4.5712,E2 449.824} C_DIS
LIN {X 137.128,Y 3.1246,Z 182,A 4.3817,B 4.4065,C 0.2089,E1 4.5712,E2 448.3773} C_DIS
LIN {X 136.9226,Y 8.1031,Z 182,A 6.6401,B 4.4069,C 0.2007,E1 4.5709,E2 446.0947} C_DIS
LIN {X 136.5458,Y 12.9852,Z 182,A 9.143,B 4.4074,C 0.189,E1 4.5702,E2 443.5315} C_DIS
LIN {X 135.8447,Y 18.9668,Z 182,A 10.6664,B 4.4071,C 0.1948,E1 4.5697,E2 442.1339} C_DIS
LIN {X 135.4994,Y 21.2917,Z 182,A 11.7057,B 4.4073,C 0.1913,E1 4.5692,E2 441.0866} C_DIS
LIN {X 135.002,Y 24.2439,Z 182,A 12.9736,B 4.4074,C 0.1876,E1 4.5686,E2 439.8157} C_DIS
LIN {X 134.3865,Y 27.4513,Z 182,A 14.3739,B 4.4076,C 0.1834,E1 4.5679,E2 438.4101} C_DIS
LIN {X 133.5975,Y 31.0692,Z 182,A 15.7905,B 4.4077,C 0.1807,E1 4.567,E2 437.0091} C_DIS
LIN {X 132.8764,Y 34.0182,Z 182,A 16.9932,B 4.4078,C 0.1781,E1 4.5662,E2 435.8139} C_DIS
LIN {X 132.0549,Y 37.0782,Z 182,A 18.332,B 4.408,C 0.1743,E1 4.5652,E2 434.4724} C_DIS
LIN {X 131.0428,Y 40.5119,Z 182,A 19.8015,B 4.4081,C 0.1706,E1 4.564,E2 433.0054} C_DIS
LIN {X 130.0308,Y 43.6503,Z 182,A 21.0718,B 4.4082,C 0.1682,E1 4.5629,E2 431.748} C_DIS
LIN {X 128.9728,Y 46.683,Z 182,A 22.4014,B 4.4084,C 0.1648,E1 4.5617,E2 430.4192} C_DIS
LIN {X 127.5322,Y 50.4926,Z 182,A 24.0471,B 4.4084,C 0.161,E1 4.56,E2 428.7798} C_DIS
LIN {X 126.6247,Y 52.7204,Z 182,A 25.1361,B 4.4086,C 0.1573,E1 4.5588,E2 427.6796} C_DIS
LIN {X 125.0158,Y 56.4313,Z 182,A 26.6522,B 4.4087,C 0.1551,E1 4.5571,E2 426.1846} C_DIS
LIN {X 123.3671,Y 59.9536,Z 182,A 28.2276,B 4.4088,C 0.1515,E1 4.5553,E2 424.6147} C_DIS
LIN {X 121.9359,Y 62.8115,Z 182,A 29.5758,B 4.409,C 0.148,E1 4.5535,E2 423.2643} C_DIS
LIN {X 119.9179,Y 66.5845,Z 182,A 31.3708,B 4.4091,C 0.1434,E1 4.5511,E2 421.4676} C_DIS
LIN {X 117.63,Y 70.5486,Z 182,A 33.2457,B 4.4092,C 0.1392,E1 4.5485,E2 419.5967} C_DIS
LIN {X 115.2771,Y 74.3314,Z 182,A 35.0361,B 4.4093,C 0.1356,E1 4.5458,E2 417.8145} C_DIS
LIN {X 112.8211,Y 78.0085,Z 182,A 36.7982,B 4.4094,C 0.1323,E1 4.5431,E2 416.0625} C_DIS
LIN {X 110.6041,Y 81.1204,Z 182,A 38.401,B 4.4096,C 0.1285,E1 4.5404,E2 414.4583} C_DIS
LIN {X 107.6038,Y 85.061,Z 182,A 40.3118,B 4.4096,C 0.1257,E1 4.5372,E2 412.5667} C_DIS
LIN {X 105.0732,Y 88.1668,Z 182,A 41.8513,B 4.4096,C 0.1237,E1 4.5345,E2 411.0435} C_DIS
LIN {X 102.6944,Y 90.9266,Z 182,A 43.5214,B 4.4098,C 0.1186,E1 4.5314,E2 409.3546} C_DIS
LIN {X 99.427,Y 94.4891,Z 182,A 45.3773,B 4.4098,C 0.1163,E1 4.5279,E2 407.5187} C_DIS
LIN {X 96.9328,Y 97.046,Z 182,A 46.9844,B 4.41,C 0.1119,E1 4.5247,E2 405.8969} C_DIS
LIN {X 93.0105,Y 100.8111,Z 182,A 49.0516,B 4.41,C 0.1098,E1 4.5206,E2 403.8548} C_DIS
LIN {X 90.0493,Y 103.4646,Z 182,A 50.7565,B 4.4102,C 0.1061,E1 4.517,E2 402.1442} C_DIS
LIN {X 86.6879,Y 106.2968,Z 182,A 52.5454,B 4.4102,C 0.1033,E1 4.5132,E2 400.3609} C_DIS
LIN {X 83.8185,Y 108.5739,Z 182,A 54.0537,B 4.4102,C 0.1008,E1 4.5099,E2 398.8552} C_DIS
LIN {X 80.7048,Y 110.908,Z 182,A 55.7118,B 4.4103,C 0.0976,E1 4.5061,E2 397.1929} C_DIS
LIN {X 76.9929,Y 113.516,Z 182,A 57.5642,B 4.4104,C 0.095,E1 4.5019,E2 395.3457} C_DIS
LIN {X 73.066,Y 116.0826,Z 182,A 59.4753,B 4.4104,C 0.0925,E1 4.4974,E2 393.4407} C_DIS
LIN {X 69.1112,Y 118.4804,Z 182,A 61.4112,B 4.4105,C 0.0895,E1 4.4927,E2 391.5044} C_DIS
LIN {X 65.3008,Y 120.6224,Z 182,A 63.212,B 4.4105,C 0.0872,E1 4.4883,E2 389.7068} C_DIS
LIN {X 62.0084,Y 122.3448,Z 182,A 64.6109,B 4.4105,C 0.0868,E1 4.4849,E2 388.3268} C_DIS
LIN {X 59.2145,Y 123.721,Z 182,A 65.9492,B 4.4106,C 0.0848,E1 4.4815,E2 386.984} C_DIS
LIN {X 55.7577,Y 125.3171,Z 182,A 67.4546,B 4.4106,C 0.0837,E1 4.4777,E2 385.4894} C_DIS
LIN {X 52.8859,Y 126.5556,Z 182,A 68.8088,B 4.4106,C 0.0817,E1 4.4742,E2 384.1294} C_DIS
LIN {X 49.3918,Y 127.9602,Z 182,A 70.2566,B 4.4106,C 0.0813,E1 4.4705,E2 382.6973} C_DIS
LIN {X 46.4356,Y 129.062,Z 182,A 71.6233,B 4.4107,C 0.0794,E1 4.4669,E2 381.3248} C_DIS
LIN {X 42.9961,Y 130.2487,Z 182,A 73.1053,B 4.4107,C 0.0784,E1 4.463,E2 379.8477} C_DIS
LIN {X 40.0919,Y 131.1713,Z 182,A 74.451,B 4.4107,C 0.0765,E1 4.4594,E2 378.4933} C_DIS
LIN {X 36.4785,Y 132.2226,Z 182,A 75.8843,B 4.4107,C 0.0766,E1 4.4556,E2 377.0775} C_DIS
LIN {X 33.5237,Y 133.0019,Z 182,A 77.2071,B 4.4107,C 0.0752,E1 4.452,E2 375.7493} C_DIS
LIN {X 29.3375,Y 133.988,Z 182,A 79.0075,B 4.4108,C 0.0739,E1 4.4471,E2 373.9489} C_DIS
LIN {X 25.8477,Y 134.7042,Z 182,A 80.4689,B 4.4108,C 0.0732,E1 4.4431,E2 372.4912} C_DIS
LIN {X 22.579,Y 135.2904,Z 182,A 81.8247,B 4.4108,C 0.0728,E1 4.4394,E2 371.1398} C_DIS
LIN {X 19.2094,Y 135.81,Z 182,A 83.5948,B 4.4108,C 0.0686,E1 4.4343,E2 369.3275} C_DIS
LIN {X 15.4848,Y 136.287,Z 182,A 85.3582,B 4.4109,C 0.0661,E1 4.4294,E2 367.5406} C_DIS
LIN {X 10.8564,Y 136.7328,Z 182,A 86.6989,B 4.4109,C 0.0715,E1 4.4259,E2 366.2749} C_DIS
LIN {X 5.6819,Y 137.0445,Z 182,A 88.9515,B 4.4109,C 0.0701,E1 4.4195,E2 364.0124} C_DIS
LIN {X 2.3258,Y 137.1422,Z 182,A 90.2691,B 4.4109,C 0.0708,E1 4.4159,E2 362.7057} C_DIS
LIN {X -0.2391,Y 137.1627,Z 182,A 91.4648,B 4.4109,C 0.0695,E1 4.4125,E2 361.4954} C_DIS
LIN {X -4.1046,Y 137.1008,Z 182,A 93.0583,B 4.4109,C 0.0697,E1 4.4081,E2 359.9052} C_DIS
LIN {X -7.6487,Y 136.9505,Z 182,A 94.448,B 4.4109,C 0.0707,E1 4.4042,E2 358.5276} C_DIS
LIN {X -11.5392,Y 136.6755,Z 182,A 96.7858,B 4.4109,C 0.0643,E1 4.3975,E2 356.1031} C_DIS
LIN {X -16.9868,Y 136.1078,Z 182,A 98.3678,B 4.4109,C 0.0715,E1 4.3933,E2 354.6094} C_DIS
LIN {X -19.6564,Y 135.7462,Z 182,A 99.577,B 4.4109,C 0.0711,E1 4.39,E2 353.3905} C_DIS
LIN {X -23.1564,Y 135.1941,Z 182,A 100.9788,B 4.4109,C 0.0724,E1 4.3861,E2 351.9991} C_DIS
LIN {X -25.7681,Y 134.7194,Z 182,A 102.1959,B 4.4109,C 0.0719,E1 4.3827,E2 350.7694} C_DIS
Enddeposition()
END
